   AxisStore[3].Axis[12].Pos24.Reached := FALSE;
   AxisStore[3].Axis[12].Pos25.Position := 0.0;
   AxisStore[3].Axis[12].Pos25.Speed := 0;
   AxisStore[3].Axis[12].Pos25.Reached := FALSE;
   AxisStore[3].Axis[12].Pos26.Position := 0.0;
   AxisStore[3].Axis[12].Pos26.Speed := 0;
   AxisStore[3].Axis[12].Pos26.Reached := FALSE;
   AxisStore[3].Axis[12].Pos27.Position := 0.0;
   AxisStore[3].Axis[12].Pos27.Speed := 0;
   AxisStore[3].Axis[12].Pos27.Reached := FALSE;
   AxisStore[3].Axis[12].Pos28.Position := 0.0;
   AxisStore[3].Axis[12].Pos28.Speed := 0;
   AxisStore[3].Axis[12].Pos28.Reached := FALSE;
   AxisStore[3].Axis[12].Pos29.Position := 0.0;
   AxisStore[3].Axis[12].Pos29.Speed := 0;
   AxisStore[3].Axis[12].Pos29.Reached := FALSE;
   AxisStore[3].Axis[12].Pos30.Position := 0.0;
   AxisStore[3].Axis[12].Pos30.Speed := 0;
   AxisStore[3].Axis[12].Pos30.Reached := FALSE;
   AxisStore[3].Axis[13].Pos1.Position := 0.0;
   AxisStore[3].Axis[13].Pos1.Speed := 0;
   AxisStore[3].Axis[13].Pos1.Reached := FALSE;
   AxisStore[3].Axis[13].Pos2.Position := 0.0;
   AxisStore[3].Axis[13].Pos2.Speed := 0;
   AxisStore[3].Axis[13].Pos2.Reached := FALSE;
   AxisStore[3].Axis[13].Pos3.Position := 0.0;
   AxisStore[3].Axis[13].Pos3.Speed := 0;
   AxisStore[3].Axis[13].Pos3.Reached := FALSE;
   AxisStore[3].Axis[13].Pos4.Position := 0.0;
   AxisStore[3].Axis[13].Pos4.Speed := 0;
   AxisStore[3].Axis[13].Pos4.Reached := FALSE;
   AxisStore[3].Axis[13].Pos5.Position := 0.0;
   AxisStore[3].Axis[13].Pos5.Speed := 0;
   AxisStore[3].Axis[13].Pos5.Reached := FALSE;
   AxisStore[3].Axis[13].Pos6.Position := 0.0;
   AxisStore[3].Axis[13].Pos6.Speed := 0;
   AxisStore[3].Axis[13].Pos6.Reached := FALSE;
   AxisStore[3].Axis[13].Pos7.Position := 0.0;
   AxisStore[3].Axis[13].Pos7.Speed := 0;
   AxisStore[3].Axis[13].Pos7.Reached := FALSE;
   AxisStore[3].Axis[13].Pos8.Position := 0.0;
   AxisStore[3].Axis[13].Pos8.Speed := 0;
   AxisStore[3].Axis[13].Pos8.Reached := FALSE;
   AxisStore[3].Axis[13].Pos9.Position := 0.0;
   AxisStore[3].Axis[13].Pos9.Speed := 0;
   AxisStore[3].Axis[13].Pos9.Reached := FALSE;
   AxisStore[3].Axis[13].Pos10.Position := 0.0;
   AxisStore[3].Axis[13].Pos10.Speed := 0;
   AxisStore[3].Axis[13].Pos10.Reached := FALSE;
   AxisStore[3].Axis[13].Pos11.Position := 0.0;
   AxisStore[3].Axis[13].Pos11.Speed := 0;
   AxisStore[3].Axis[13].Pos11.Reached := FALSE;
   AxisStore[3].Axis[13].Pos12.Position := 0.0;
   AxisStore[3].Axis[13].Pos12.Speed := 0;
   AxisStore[3].Axis[13].Pos12.Reached := FALSE;
   AxisStore[3].Axis[13].Pos13.Position := 0.0;
   AxisStore[3].Axis[13].Pos13.Speed := 0;
   AxisStore[3].Axis[13].Pos13.Reached := FALSE;
   AxisStore[3].Axis[13].Pos14.Position := 0.0;
   AxisStore[3].Axis[13].Pos14.Speed := 0;
   AxisStore[3].Axis[13].Pos14.Reached := FALSE;
   AxisStore[3].Axis[13].Pos15.Position := 0.0;
   AxisStore[3].Axis[13].Pos15.Speed := 0;
   AxisStore[3].Axis[13].Pos15.Reached := FALSE;
   AxisStore[3].Axis[13].Pos16.Position := 0.0;
   AxisStore[3].Axis[13].Pos16.Speed := 0;
   AxisStore[3].Axis[13].Pos16.Reached := FALSE;
   AxisStore[3].Axis[13].Pos17.Position := 0.0;
   AxisStore[3].Axis[13].Pos17.Speed := 0;
   AxisStore[3].Axis[13].Pos17.Reached := FALSE;
   AxisStore[3].Axis[13].Pos18.Position := 0.0;
   AxisStore[3].Axis[13].Pos18.Speed := 0;
   AxisStore[3].Axis[13].Pos18.Reached := FALSE;
   AxisStore[3].Axis[13].Pos19.Position := 0.0;
   AxisStore[3].Axis[13].Pos19.Speed := 0;
   AxisStore[3].Axis[13].Pos19.Reached := FALSE;
   AxisStore[3].Axis[13].Pos20.Position := 0.0;
   AxisStore[3].Axis[13].Pos20.Speed := 0;
   AxisStore[3].Axis[13].Pos20.Reached := FALSE;
   AxisStore[3].Axis[13].Pos21.Position := 0.0;
   AxisStore[3].Axis[13].Pos21.Speed := 0;
   AxisStore[3].Axis[13].Pos21.Reached := FALSE;
   AxisStore[3].Axis[13].Pos22.Position := 0.0;
   AxisStore[3].Axis[13].Pos22.Speed := 0;
   AxisStore[3].Axis[13].Pos22.Reached := FALSE;
   AxisStore[3].Axis[13].Pos23.Position := 0.0;
   AxisStore[3].Axis[13].Pos23.Speed := 0;
   AxisStore[3].Axis[13].Pos23.Reached := FALSE;
   AxisStore[3].Axis[13].Pos24.Position := 0.0;
   AxisStore[3].Axis[13].Pos24.Speed := 0;
   AxisStore[3].Axis[13].Pos24.Reached := FALSE;
   AxisStore[3].Axis[13].Pos25.Position := 0.0;
   AxisStore[3].Axis[13].Pos25.Speed := 0;
   AxisStore[3].Axis[13].Pos25.Reached := FALSE;
   AxisStore[3].Axis[13].Pos26.Position := 0.0;
   AxisStore[3].Axis[13].Pos26.Speed := 0;
   AxisStore[3].Axis[13].Pos26.Reached := FALSE;
   AxisStore[3].Axis[13].Pos27.Position := 0.0;
   AxisStore[3].Axis[13].Pos27.Speed := 0;
   AxisStore[3].Axis[13].Pos27.Reached := FALSE;
   AxisStore[3].Axis[13].Pos28.Position := 0.0;
   AxisStore[3].Axis[13].Pos28.Speed := 0;
   AxisStore[3].Axis[13].Pos28.Reached := FALSE;
   AxisStore[3].Axis[13].Pos29.Position := 0.0;
   AxisStore[3].Axis[13].Pos29.Speed := 0;
   AxisStore[3].Axis[13].Pos29.Reached := FALSE;
   AxisStore[3].Axis[13].Pos30.Position := 0.0;
   AxisStore[3].Axis[13].Pos30.Speed := 0;
   AxisStore[3].Axis[13].Pos30.Reached := FALSE;
   AxisStore[3].Axis[14].Pos1.Position := 0.0;
   AxisStore[3].Axis[14].Pos1.Speed := 0;
   AxisStore[3].Axis[14].Pos1.Reached := FALSE;
   AxisStore[3].Axis[14].Pos2.Position := 0.0;
   AxisStore[3].Axis[14].Pos2.Speed := 0;
   AxisStore[3].Axis[14].Pos2.Reached := FALSE;
   AxisStore[3].Axis[14].Pos3.Position := 0.0;
   AxisStore[3].Axis[14].Pos3.Speed := 0;
   AxisStore[3].Axis[14].Pos3.Reached := FALSE;
   AxisStore[3].Axis[14].Pos4.Position := 0.0;
   AxisStore[3].Axis[14].Pos4.Speed := 0;
   AxisStore[3].Axis[14].Pos4.Reached := FALSE;
   AxisStore[3].Axis[14].Pos5.Position := 0.0;
   AxisStore[3].Axis[14].Pos5.Speed := 0;
   AxisStore[3].Axis[14].Pos5.Reached := FALSE;
   AxisStore[3].Axis[14].Pos6.Position := 0.0;
   AxisStore[3].Axis[14].Pos6.Speed := 0;
   AxisStore[3].Axis[14].Pos6.Reached := FALSE;
   AxisStore[3].Axis[14].Pos7.Position := 0.0;
   AxisStore[3].Axis[14].Pos7.Speed := 0;
   AxisStore[3].Axis[14].Pos7.Reached := FALSE;
   AxisStore[3].Axis[14].Pos8.Position := 0.0;
   AxisStore[3].Axis[14].Pos8.Speed := 0;
   AxisStore[3].Axis[14].Pos8.Reached := FALSE;
   AxisStore[3].Axis[14].Pos9.Position := 0.0;
   AxisStore[3].Axis[14].Pos9.Speed := 0;
   AxisStore[3].Axis[14].Pos9.Reached := FALSE;
   AxisStore[3].Axis[14].Pos10.Position := 0.0;
   AxisStore[3].Axis[14].Pos10.Speed := 0;
   AxisStore[3].Axis[14].Pos10.Reached := FALSE;
   AxisStore[3].Axis[14].Pos11.Position := 0.0;
   AxisStore[3].Axis[14].Pos11.Speed := 0;
   AxisStore[3].Axis[14].Pos11.Reached := FALSE;
   AxisStore[3].Axis[14].Pos12.Position := 0.0;
   AxisStore[3].Axis[14].Pos12.Speed := 0;
   AxisStore[3].Axis[14].Pos12.Reached := FALSE;
   AxisStore[3].Axis[14].Pos13.Position := 0.0;
   AxisStore[3].Axis[14].Pos13.Speed := 0;
   AxisStore[3].Axis[14].Pos13.Reached := FALSE;
   AxisStore[3].Axis[14].Pos14.Position := 0.0;
   AxisStore[3].Axis[14].Pos14.Speed := 0;
   AxisStore[3].Axis[14].Pos14.Reached := FALSE;
   AxisStore[3].Axis[14].Pos15.Position := 0.0;
   AxisStore[3].Axis[14].Pos15.Speed := 0;
   AxisStore[3].Axis[14].Pos15.Reached := FALSE;
   AxisStore[3].Axis[14].Pos16.Position := 0.0;
   AxisStore[3].Axis[14].Pos16.Speed := 0;
   AxisStore[3].Axis[14].Pos16.Reached := FALSE;
   AxisStore[3].Axis[14].Pos17.Position := 0.0;
   AxisStore[3].Axis[14].Pos17.Speed := 0;
   AxisStore[3].Axis[14].Pos17.Reached := FALSE;
   AxisStore[3].Axis[14].Pos18.Position := 0.0;
   AxisStore[3].Axis[14].Pos18.Speed := 0;
   AxisStore[3].Axis[14].Pos18.Reached := FALSE;
   AxisStore[3].Axis[14].Pos19.Position := 0.0;
   AxisStore[3].Axis[14].Pos19.Speed := 0;
   AxisStore[3].Axis[14].Pos19.Reached := FALSE;
   AxisStore[3].Axis[14].Pos20.Position := 0.0;
   AxisStore[3].Axis[14].Pos20.Speed := 0;
   AxisStore[3].Axis[14].Pos20.Reached := FALSE;
   AxisStore[3].Axis[14].Pos21.Position := 0.0;
   AxisStore[3].Axis[14].Pos21.Speed := 0;
   AxisStore[3].Axis[14].Pos21.Reached := FALSE;
   AxisStore[3].Axis[14].Pos22.Position := 0.0;
   AxisStore[3].Axis[14].Pos22.Speed := 0;
   AxisStore[3].Axis[14].Pos22.Reached := FALSE;
   AxisStore[3].Axis[14].Pos23.Position := 0.0;
   AxisStore[3].Axis[14].Pos23.Speed := 0;
   AxisStore[3].Axis[14].Pos23.Reached := FALSE;
   AxisStore[3].Axis[14].Pos24.Position := 0.0;
   AxisStore[3].Axis[14].Pos24.Speed := 0;
   AxisStore[3].Axis[14].Pos24.Reached := FALSE;
   AxisStore[3].Axis[14].Pos25.Position := 0.0;
   AxisStore[3].Axis[14].Pos25.Speed := 0;
   AxisStore[3].Axis[14].Pos25.Reached := FALSE;
   AxisStore[3].Axis[14].Pos26.Position := 0.0;
   AxisStore[3].Axis[14].Pos26.Speed := 0;
   AxisStore[3].Axis[14].Pos26.Reached := FALSE;
   AxisStore[3].Axis[14].Pos27.Position := 0.0;
   AxisStore[3].Axis[14].Pos27.Speed := 0;
   AxisStore[3].Axis[14].Pos27.Reached := FALSE;
   AxisStore[3].Axis[14].Pos28.Position := 0.0;
   AxisStore[3].Axis[14].Pos28.Speed := 0;
   AxisStore[3].Axis[14].Pos28.Reached := FALSE;
   AxisStore[3].Axis[14].Pos29.Position := 0.0;
   AxisStore[3].Axis[14].Pos29.Speed := 0;
   AxisStore[3].Axis[14].Pos29.Reached := FALSE;
   AxisStore[3].Axis[14].Pos30.Position := 0.0;
   AxisStore[3].Axis[14].Pos30.Speed := 0;
   AxisStore[3].Axis[14].Pos30.Reached := FALSE;
   AxisStore[3].Axis[15].Pos1.Position := 0.0;
   AxisStore[3].Axis[15].Pos1.Speed := 0;
   AxisStore[3].Axis[15].Pos1.Reached := FALSE;
   AxisStore[3].Axis[15].Pos2.Position := 0.0;
   AxisStore[3].Axis[15].Pos2.Speed := 0;
   AxisStore[3].Axis[15].Pos2.Reached := FALSE;
   AxisStore[3].Axis[15].Pos3.Position := 0.0;
   AxisStore[3].Axis[15].Pos3.Speed := 0;
   AxisStore[3].Axis[15].Pos3.Reached := FALSE;
   AxisStore[3].Axis[15].Pos4.Position := 0.0;
   AxisStore[3].Axis[15].Pos4.Speed := 0;
   AxisStore[3].Axis[15].Pos4.Reached := FALSE;
   AxisStore[3].Axis[15].Pos5.Position := 0.0;
   AxisStore[3].Axis[15].Pos5.Speed := 0;
   AxisStore[3].Axis[15].Pos5.Reached := FALSE;
   AxisStore[3].Axis[15].Pos6.Position := 0.0;
   AxisStore[3].Axis[15].Pos6.Speed := 0;
   AxisStore[3].Axis[15].Pos6.Reached := FALSE;
   AxisStore[3].Axis[15].Pos7.Position := 0.0;
   AxisStore[3].Axis[15].Pos7.Speed := 0;
   AxisStore[3].Axis[15].Pos7.Reached := FALSE;
   AxisStore[3].Axis[15].Pos8.Position := 0.0;
   AxisStore[3].Axis[15].Pos8.Speed := 0;
   AxisStore[3].Axis[15].Pos8.Reached := FALSE;
   AxisStore[3].Axis[15].Pos9.Position := 0.0;
   AxisStore[3].Axis[15].Pos9.Speed := 0;
   AxisStore[3].Axis[15].Pos9.Reached := FALSE;
   AxisStore[3].Axis[15].Pos10.Position := 0.0;
   AxisStore[3].Axis[15].Pos10.Speed := 0;
   AxisStore[3].Axis[15].Pos10.Reached := FALSE;
   AxisStore[3].Axis[15].Pos11.Position := 0.0;
   AxisStore[3].Axis[15].Pos11.Speed := 0;
   AxisStore[3].Axis[15].Pos11.Reached := FALSE;
   AxisStore[3].Axis[15].Pos12.Position := 0.0;
   AxisStore[3].Axis[15].Pos12.Speed := 0;
   AxisStore[3].Axis[15].Pos12.Reached := FALSE;
   AxisStore[3].Axis[15].Pos13.Position := 0.0;
   AxisStore[3].Axis[15].Pos13.Speed := 0;
   AxisStore[3].Axis[15].Pos13.Reached := FALSE;
   AxisStore[3].Axis[15].Pos14.Position := 0.0;
   AxisStore[3].Axis[15].Pos14.Speed := 0;
   AxisStore[3].Axis[15].Pos14.Reached := FALSE;
   AxisStore[3].Axis[15].Pos15.Position := 0.0;
   AxisStore[3].Axis[15].Pos15.Speed := 0;
   AxisStore[3].Axis[15].Pos15.Reached := FALSE;
   AxisStore[3].Axis[15].Pos16.Position := 0.0;
   AxisStore[3].Axis[15].Pos16.Speed := 0;
   AxisStore[3].Axis[15].Pos16.Reached := FALSE;
   AxisStore[3].Axis[15].Pos17.Position := 0.0;
   AxisStore[3].Axis[15].Pos17.Speed := 0;
   AxisStore[3].Axis[15].Pos17.Reached := FALSE;
   AxisStore[3].Axis[15].Pos18.Position := 0.0;
   AxisStore[3].Axis[15].Pos18.Speed := 0;
   AxisStore[3].Axis[15].Pos18.Reached := FALSE;
   AxisStore[3].Axis[15].Pos19.Position := 0.0;
   AxisStore[3].Axis[15].Pos19.Speed := 0;
   AxisStore[3].Axis[15].Pos19.Reached := FALSE;
   AxisStore[3].Axis[15].Pos20.Position := 0.0;
   AxisStore[3].Axis[15].Pos20.Speed := 0;
   AxisStore[3].Axis[15].Pos20.Reached := FALSE;
   AxisStore[3].Axis[15].Pos21.Position := 0.0;
   AxisStore[3].Axis[15].Pos21.Speed := 0;
   AxisStore[3].Axis[15].Pos21.Reached := FALSE;
   AxisStore[3].Axis[15].Pos22.Position := 0.0;
   AxisStore[3].Axis[15].Pos22.Speed := 0;
   AxisStore[3].Axis[15].Pos22.Reached := FALSE;
   AxisStore[3].Axis[15].Pos23.Position := 0.0;
   AxisStore[3].Axis[15].Pos23.Speed := 0;
   AxisStore[3].Axis[15].Pos23.Reached := FALSE;
   AxisStore[3].Axis[15].Pos24.Position := 0.0;
   AxisStore[3].Axis[15].Pos24.Speed := 0;
   AxisStore[3].Axis[15].Pos24.Reached := FALSE;
   AxisStore[3].Axis[15].Pos25.Position := 0.0;
   AxisStore[3].Axis[15].Pos25.Speed := 0;
   AxisStore[3].Axis[15].Pos25.Reached := FALSE;
   AxisStore[3].Axis[15].Pos26.Position := 0.0;
   AxisStore[3].Axis[15].Pos26.Speed := 0;
   AxisStore[3].Axis[15].Pos26.Reached := FALSE;
   AxisStore[3].Axis[15].Pos27.Position := 0.0;
   AxisStore[3].Axis[15].Pos27.Speed := 0;
   AxisStore[3].Axis[15].Pos27.Reached := FALSE;
   AxisStore[3].Axis[15].Pos28.Position := 0.0;
   AxisStore[3].Axis[15].Pos28.Speed := 0;
   AxisStore[3].Axis[15].Pos28.Reached := FALSE;
   AxisStore[3].Axis[15].Pos29.Position := 0.0;
   AxisStore[3].Axis[15].Pos29.Speed := 0;
   AxisStore[3].Axis[15].Pos29.Reached := FALSE;
   AxisStore[3].Axis[15].Pos30.Position := 0.0;
   AxisStore[3].Axis[15].Pos30.Speed := 0;
   AxisStore[3].Axis[15].Pos30.Reached := FALSE;
   AxisStore[4].Axis[1].Pos1.Position := 0.0;
   AxisStore[4].Axis[1].Pos1.Speed := 0;
   AxisStore[4].Axis[1].Pos1.Reached := FALSE;
   AxisStore[4].Axis[1].Pos2.Position := 0.0;
   AxisStore[4].Axis[1].Pos2.Speed := 0;
   AxisStore[4].Axis[1].Pos2.Reached := FALSE;
   AxisStore[4].Axis[1].Pos3.Position := 0.0;
   AxisStore[4].Axis[1].Pos3.Speed := 0;
   AxisStore[4].Axis[1].Pos3.Reached := FALSE;
   AxisStore[4].Axis[1].Pos4.Position := 0.0;
   AxisStore[4].Axis[1].Pos4.Speed := 0;
   AxisStore[4].Axis[1].Pos4.Reached := FALSE;
   AxisStore[4].Axis[1].Pos5.Position := 0.0;
   AxisStore[4].Axis[1].Pos5.Speed := 0;
   AxisStore[4].Axis[1].Pos5.Reached := FALSE;
   AxisStore[4].Axis[1].Pos6.Position := 0.0;
   AxisStore[4].Axis[1].Pos6.Speed := 0;
   AxisStore[4].Axis[1].Pos6.Reached := FALSE;
   AxisStore[4].Axis[1].Pos7.Position := 0.0;
   AxisStore[4].Axis[1].Pos7.Speed := 0;
   AxisStore[4].Axis[1].Pos7.Reached := FALSE;
   AxisStore[4].Axis[1].Pos8.Position := 0.0;
   AxisStore[4].Axis[1].Pos8.Speed := 0;
   AxisStore[4].Axis[1].Pos8.Reached := FALSE;
   AxisStore[4].Axis[1].Pos9.Position := 0.0;
   AxisStore[4].Axis[1].Pos9.Speed := 0;
   AxisStore[4].Axis[1].Pos9.Reached := FALSE;
   AxisStore[4].Axis[1].Pos10.Position := 0.0;
   AxisStore[4].Axis[1].Pos10.Speed := 0;
   AxisStore[4].Axis[1].Pos10.Reached := FALSE;
   AxisStore[4].Axis[1].Pos11.Position := 0.0;
   AxisStore[4].Axis[1].Pos11.Speed := 0;
   AxisStore[4].Axis[1].Pos11.Reached := FALSE;
   AxisStore[4].Axis[1].Pos12.Position := 0.0;
   AxisStore[4].Axis[1].Pos12.Speed := 0;
   AxisStore[4].Axis[1].Pos12.Reached := FALSE;
   AxisStore[4].Axis[1].Pos13.Position := 0.0;
   AxisStore[4].Axis[1].Pos13.Speed := 0;
   AxisStore[4].Axis[1].Pos13.Reached := FALSE;
   AxisStore[4].Axis[1].Pos14.Position := 0.0;
   AxisStore[4].Axis[1].Pos14.Speed := 0;
   AxisStore[4].Axis[1].Pos14.Reached := FALSE;
   AxisStore[4].Axis[1].Pos15.Position := 0.0;
   AxisStore[4].Axis[1].Pos15.Speed := 0;
   AxisStore[4].Axis[1].Pos15.Reached := FALSE;
   AxisStore[4].Axis[1].Pos16.Position := 0.0;
   AxisStore[4].Axis[1].Pos16.Speed := 0;
   AxisStore[4].Axis[1].Pos16.Reached := FALSE;
   AxisStore[4].Axis[1].Pos17.Position := 0.0;
   AxisStore[4].Axis[1].Pos17.Speed := 0;
   AxisStore[4].Axis[1].Pos17.Reached := FALSE;
   AxisStore[4].Axis[1].Pos18.Position := 0.0;
   AxisStore[4].Axis[1].Pos18.Speed := 0;
   AxisStore[4].Axis[1].Pos18.Reached := FALSE;
   AxisStore[4].Axis[1].Pos19.Position := 0.0;
   AxisStore[4].Axis[1].Pos19.Speed := 0;
   AxisStore[4].Axis[1].Pos19.Reached := FALSE;
   AxisStore[4].Axis[1].Pos20.Position := 0.0;
   AxisStore[4].Axis[1].Pos20.Speed := 0;
   AxisStore[4].Axis[1].Pos20.Reached := FALSE;
   AxisStore[4].Axis[1].Pos21.Position := 0.0;
   AxisStore[4].Axis[1].Pos21.Speed := 0;
   AxisStore[4].Axis[1].Pos21.Reached := FALSE;
   AxisStore[4].Axis[1].Pos22.Position := 0.0;
   AxisStore[4].Axis[1].Pos22.Speed := 0;
   AxisStore[4].Axis[1].Pos22.Reached := FALSE;
   AxisStore[4].Axis[1].Pos23.Position := 0.0;
   AxisStore[4].Axis[1].Pos23.Speed := 0;
   AxisStore[4].Axis[1].Pos23.Reached := FALSE;
   AxisStore[4].Axis[1].Pos24.Position := 0.0;
   AxisStore[4].Axis[1].Pos24.Speed := 0;
   AxisStore[4].Axis[1].Pos24.Reached := FALSE;
   AxisStore[4].Axis[1].Pos25.Position := 0.0;
   AxisStore[4].Axis[1].Pos25.Speed := 0;
   AxisStore[4].Axis[1].Pos25.Reached := FALSE;
   AxisStore[4].Axis[1].Pos26.Position := 0.0;
   AxisStore[4].Axis[1].Pos26.Speed := 0;
   AxisStore[4].Axis[1].Pos26.Reached := FALSE;
   AxisStore[4].Axis[1].Pos27.Position := 0.0;
   AxisStore[4].Axis[1].Pos27.Speed := 0;
   AxisStore[4].Axis[1].Pos27.Reached := FALSE;
   AxisStore[4].Axis[1].Pos28.Position := 0.0;
   AxisStore[4].Axis[1].Pos28.Speed := 0;
   AxisStore[4].Axis[1].Pos28.Reached := FALSE;
   AxisStore[4].Axis[1].Pos29.Position := 0.0;
   AxisStore[4].Axis[1].Pos29.Speed := 0;
   AxisStore[4].Axis[1].Pos29.Reached := FALSE;
   AxisStore[4].Axis[1].Pos30.Position := 0.0;
   AxisStore[4].Axis[1].Pos30.Speed := 0;
   AxisStore[4].Axis[1].Pos30.Reached := FALSE;
   AxisStore[4].Axis[2].Pos1.Position := 0.0;
   AxisStore[4].Axis[2].Pos1.Speed := 0;
   AxisStore[4].Axis[2].Pos1.Reached := FALSE;
   AxisStore[4].Axis[2].Pos2.Position := 0.0;
   AxisStore[4].Axis[2].Pos2.Speed := 0;
   AxisStore[4].Axis[2].Pos2.Reached := FALSE;
   AxisStore[4].Axis[2].Pos3.Position := 0.0;
   AxisStore[4].Axis[2].Pos3.Speed := 0;
   AxisStore[4].Axis[2].Pos3.Reached := FALSE;
   AxisStore[4].Axis[2].Pos4.Position := 0.0;
   AxisStore[4].Axis[2].Pos4.Speed := 0;
   AxisStore[4].Axis[2].Pos4.Reached := FALSE;
   AxisStore[4].Axis[2].Pos5.Position := 0.0;
   AxisStore[4].Axis[2].Pos5.Speed := 0;
   AxisStore[4].Axis[2].Pos5.Reached := FALSE;
   AxisStore[4].Axis[2].Pos6.Position := 0.0;
   AxisStore[4].Axis[2].Pos6.Speed := 0;
   AxisStore[4].Axis[2].Pos6.Reached := FALSE;
   AxisStore[4].Axis[2].Pos7.Position := 0.0;
   AxisStore[4].Axis[2].Pos7.Speed := 0;
   AxisStore[4].Axis[2].Pos7.Reached := FALSE;
   AxisStore[4].Axis[2].Pos8.Position := 0.0;
   AxisStore[4].Axis[2].Pos8.Speed := 0;
   AxisStore[4].Axis[2].Pos8.Reached := FALSE;
   AxisStore[4].Axis[2].Pos9.Position := 0.0;
   AxisStore[4].Axis[2].Pos9.Speed := 0;
   AxisStore[4].Axis[2].Pos9.Reached := FALSE;
   AxisStore[4].Axis[2].Pos10.Position := 0.0;
   AxisStore[4].Axis[2].Pos10.Speed := 0;
   AxisStore[4].Axis[2].Pos10.Reached := FALSE;
   AxisStore[4].Axis[2].Pos11.Position := 0.0;
   AxisStore[4].Axis[2].Pos11.Speed := 0;
   AxisStore[4].Axis[2].Pos11.Reached := FALSE;
   AxisStore[4].Axis[2].Pos12.Position := 0.0;
   AxisStore[4].Axis[2].Pos12.Speed := 0;
   AxisStore[4].Axis[2].Pos12.Reached := FALSE;
   AxisStore[4].Axis[2].Pos13.Position := 0.0;
   AxisStore[4].Axis[2].Pos13.Speed := 0;
   AxisStore[4].Axis[2].Pos13.Reached := FALSE;
   AxisStore[4].Axis[2].Pos14.Position := 0.0;
   AxisStore[4].Axis[2].Pos14.Speed := 0;
   AxisStore[4].Axis[2].Pos14.Reached := FALSE;
   AxisStore[4].Axis[2].Pos15.Position := 0.0;
   AxisStore[4].Axis[2].Pos15.Speed := 0;
   AxisStore[4].Axis[2].Pos15.Reached := FALSE;
   AxisStore[4].Axis[2].Pos16.Position := 0.0;
   AxisStore[4].Axis[2].Pos16.Speed := 0;
   AxisStore[4].Axis[2].Pos16.Reached := FALSE;
   AxisStore[4].Axis[2].Pos17.Position := 0.0;
   AxisStore[4].Axis[2].Pos17.Speed := 0;
   AxisStore[4].Axis[2].Pos17.Reached := FALSE;
   AxisStore[4].Axis[2].Pos18.Position := 0.0;
   AxisStore[4].Axis[2].Pos18.Speed := 0;
   AxisStore[4].Axis[2].Pos18.Reached := FALSE;
   AxisStore[4].Axis[2].Pos19.Position := 0.0;
   AxisStore[4].Axis[2].Pos19.Speed := 0;
   AxisStore[4].Axis[2].Pos19.Reached := FALSE;
   AxisStore[4].Axis[2].Pos20.Position := 0.0;
   AxisStore[4].Axis[2].Pos20.Speed := 0;
   AxisStore[4].Axis[2].Pos20.Reached := FALSE;
   AxisStore[4].Axis[2].Pos21.Position := 0.0;
   AxisStore[4].Axis[2].Pos21.Speed := 0;
   AxisStore[4].Axis[2].Pos21.Reached := FALSE;
   AxisStore[4].Axis[2].Pos22.Position := 0.0;
   AxisStore[4].Axis[2].Pos22.Speed := 0;
   AxisStore[4].Axis[2].Pos22.Reached := FALSE;
   AxisStore[4].Axis[2].Pos23.Position := 0.0;
   AxisStore[4].Axis[2].Pos23.Speed := 0;
   AxisStore[4].Axis[2].Pos23.Reached := FALSE;
   AxisStore[4].Axis[2].Pos24.Position := 0.0;
   AxisStore[4].Axis[2].Pos24.Speed := 0;
   AxisStore[4].Axis[2].Pos24.Reached := FALSE;
   AxisStore[4].Axis[2].Pos25.Position := 0.0;
   AxisStore[4].Axis[2].Pos25.Speed := 0;
   AxisStore[4].Axis[2].Pos25.Reached := FALSE;
   AxisStore[4].Axis[2].Pos26.Position := 0.0;
   AxisStore[4].Axis[2].Pos26.Speed := 0;
   AxisStore[4].Axis[2].Pos26.Reached := FALSE;
   AxisStore[4].Axis[2].Pos27.Position := 0.0;
   AxisStore[4].Axis[2].Pos27.Speed := 0;
   AxisStore[4].Axis[2].Pos27.Reached := FALSE;
   AxisStore[4].Axis[2].Pos28.Position := 0.0;
   AxisStore[4].Axis[2].Pos28.Speed := 0;
   AxisStore[4].Axis[2].Pos28.Reached := FALSE;
   AxisStore[4].Axis[2].Pos29.Position := 0.0;
   AxisStore[4].Axis[2].Pos29.Speed := 0;
   AxisStore[4].Axis[2].Pos29.Reached := FALSE;
   AxisStore[4].Axis[2].Pos30.Position := 0.0;
   AxisStore[4].Axis[2].Pos30.Speed := 0;
   AxisStore[4].Axis[2].Pos30.Reached := FALSE;
   AxisStore[4].Axis[3].Pos1.Position := 0.0;
   AxisStore[4].Axis[3].Pos1.Speed := 0;
   AxisStore[4].Axis[3].Pos1.Reached := FALSE;
   AxisStore[4].Axis[3].Pos2.Position := 0.0;
   AxisStore[4].Axis[3].Pos2.Speed := 0;
   AxisStore[4].Axis[3].Pos2.Reached := FALSE;
   AxisStore[4].Axis[3].Pos3.Position := 0.0;
   AxisStore[4].Axis[3].Pos3.Speed := 0;
   AxisStore[4].Axis[3].Pos3.Reached := FALSE;
   AxisStore[4].Axis[3].Pos4.Position := 0.0;
   AxisStore[4].Axis[3].Pos4.Speed := 0;
   AxisStore[4].Axis[3].Pos4.Reached := FALSE;
   AxisStore[4].Axis[3].Pos5.Position := 0.0;
   AxisStore[4].Axis[3].Pos5.Speed := 0;
   AxisStore[4].Axis[3].Pos5.Reached := FALSE;
   AxisStore[4].Axis[3].Pos6.Position := 0.0;
   AxisStore[4].Axis[3].Pos6.Speed := 0;
   AxisStore[4].Axis[3].Pos6.Reached := FALSE;
   AxisStore[4].Axis[3].Pos7.Position := 0.0;
   AxisStore[4].Axis[3].Pos7.Speed := 0;
   AxisStore[4].Axis[3].Pos7.Reached := FALSE;
   AxisStore[4].Axis[3].Pos8.Position := 0.0;
   AxisStore[4].Axis[3].Pos8.Speed := 0;
   AxisStore[4].Axis[3].Pos8.Reached := FALSE;
   AxisStore[4].Axis[3].Pos9.Position := 0.0;
   AxisStore[4].Axis[3].Pos9.Speed := 0;
   AxisStore[4].Axis[3].Pos9.Reached := FALSE;
   AxisStore[4].Axis[3].Pos10.Position := 0.0;
   AxisStore[4].Axis[3].Pos10.Speed := 0;
   AxisStore[4].Axis[3].Pos10.Reached := FALSE;
   AxisStore[4].Axis[3].Pos11.Position := 0.0;
   AxisStore[4].Axis[3].Pos11.Speed := 0;
   AxisStore[4].Axis[3].Pos11.Reached := FALSE;
   AxisStore[4].Axis[3].Pos12.Position := 0.0;
   AxisStore[4].Axis[3].Pos12.Speed := 0;
   AxisStore[4].Axis[3].Pos12.Reached := FALSE;
   AxisStore[4].Axis[3].Pos13.Position := 0.0;
   AxisStore[4].Axis[3].Pos13.Speed := 0;
   AxisStore[4].Axis[3].Pos13.Reached := FALSE;
   AxisStore[4].Axis[3].Pos14.Position := 0.0;
   AxisStore[4].Axis[3].Pos14.Speed := 0;
   AxisStore[4].Axis[3].Pos14.Reached := FALSE;
   AxisStore[4].Axis[3].Pos15.Position := 0.0;
   AxisStore[4].Axis[3].Pos15.Speed := 0;
   AxisStore[4].Axis[3].Pos15.Reached := FALSE;
   AxisStore[4].Axis[3].Pos16.Position := 0.0;
   AxisStore[4].Axis[3].Pos16.Speed := 0;
   AxisStore[4].Axis[3].Pos16.Reached := FALSE;
   AxisStore[4].Axis[3].Pos17.Position := 0.0;
   AxisStore[4].Axis[3].Pos17.Speed := 0;
   AxisStore[4].Axis[3].Pos17.Reached := FALSE;
   AxisStore[4].Axis[3].Pos18.Position := 0.0;
   AxisStore[4].Axis[3].Pos18.Speed := 0;
   AxisStore[4].Axis[3].Pos18.Reached := FALSE;
   AxisStore[4].Axis[3].Pos19.Position := 0.0;
   AxisStore[4].Axis[3].Pos19.Speed := 0;
   AxisStore[4].Axis[3].Pos19.Reached := FALSE;
   AxisStore[4].Axis[3].Pos20.Position := 0.0;
   AxisStore[4].Axis[3].Pos20.Speed := 0;
   AxisStore[4].Axis[3].Pos20.Reached := FALSE;
   AxisStore[4].Axis[3].Pos21.Position := 0.0;
   AxisStore[4].Axis[3].Pos21.Speed := 0;
   AxisStore[4].Axis[3].Pos21.Reached := FALSE;
   AxisStore[4].Axis[3].Pos22.Position := 0.0;
   AxisStore[4].Axis[3].Pos22.Speed := 0;
   AxisStore[4].Axis[3].Pos22.Reached := FALSE;
   AxisStore[4].Axis[3].Pos23.Position := 0.0;
   AxisStore[4].Axis[3].Pos23.Speed := 0;
   AxisStore[4].Axis[3].Pos23.Reached := FALSE;
   AxisStore[4].Axis[3].Pos24.Position := 0.0;
   AxisStore[4].Axis[3].Pos24.Speed := 0;
   AxisStore[4].Axis[3].Pos24.Reached := FALSE;
   AxisStore[4].Axis[3].Pos25.Position := 0.0;
   AxisStore[4].Axis[3].Pos25.Speed := 0;
   AxisStore[4].Axis[3].Pos25.Reached := FALSE;
   AxisStore[4].Axis[3].Pos26.Position := 0.0;
   AxisStore[4].Axis[3].Pos26.Speed := 0;
   AxisStore[4].Axis[3].Pos26.Reached := FALSE;
   AxisStore[4].Axis[3].Pos27.Position := 0.0;
   AxisStore[4].Axis[3].Pos27.Speed := 0;
   AxisStore[4].Axis[3].Pos27.Reached := FALSE;
   AxisStore[4].Axis[3].Pos28.Position := 0.0;
   AxisStore[4].Axis[3].Pos28.Speed := 0;
   AxisStore[4].Axis[3].Pos28.Reached := FALSE;
   AxisStore[4].Axis[3].Pos29.Position := 0.0;
   AxisStore[4].Axis[3].Pos29.Speed := 0;
   AxisStore[4].Axis[3].Pos29.Reached := FALSE;
   AxisStore[4].Axis[3].Pos30.Position := 0.0;
   AxisStore[4].Axis[3].Pos30.Speed := 0;
   AxisStore[4].Axis[3].Pos30.Reached := FALSE;
   AxisStore[4].Axis[4].Pos1.Position := 0.0;
   AxisStore[4].Axis[4].Pos1.Speed := 0;
   AxisStore[4].Axis[4].Pos1.Reached := FALSE;
   AxisStore[4].Axis[4].Pos2.Position := 0.0;
   AxisStore[4].Axis[4].Pos2.Speed := 0;
   AxisStore[4].Axis[4].Pos2.Reached := FALSE;
   AxisStore[4].Axis[4].Pos3.Position := 0.0;
   AxisStore[4].Axis[4].Pos3.Speed := 0;
   AxisStore[4].Axis[4].Pos3.Reached := FALSE;
   AxisStore[4].Axis[4].Pos4.Position := 0.0;
   AxisStore[4].Axis[4].Pos4.Speed := 0;
   AxisStore[4].Axis[4].Pos4.Reached := FALSE;
   AxisStore[4].Axis[4].Pos5.Position := 0.0;
   AxisStore[4].Axis[4].Pos5.Speed := 0;
   AxisStore[4].Axis[4].Pos5.Reached := FALSE;
   AxisStore[4].Axis[4].Pos6.Position := 0.0;
   AxisStore[4].Axis[4].Pos6.Speed := 0;
   AxisStore[4].Axis[4].Pos6.Reached := FALSE;
   AxisStore[4].Axis[4].Pos7.Position := 0.0;
   AxisStore[4].Axis[4].Pos7.Speed := 0;
   AxisStore[4].Axis[4].Pos7.Reached := FALSE;
   AxisStore[4].Axis[4].Pos8.Position := 0.0;
   AxisStore[4].Axis[4].Pos8.Speed := 0;
   AxisStore[4].Axis[4].Pos8.Reached := FALSE;
   AxisStore[4].Axis[4].Pos9.Position := 0.0;
   AxisStore[4].Axis[4].Pos9.Speed := 0;
   AxisStore[4].Axis[4].Pos9.Reached := FALSE;
   AxisStore[4].Axis[4].Pos10.Position := 0.0;
   AxisStore[4].Axis[4].Pos10.Speed := 0;
   AxisStore[4].Axis[4].Pos10.Reached := FALSE;
   AxisStore[4].Axis[4].Pos11.Position := 0.0;
   AxisStore[4].Axis[4].Pos11.Speed := 0;
   AxisStore[4].Axis[4].Pos11.Reached := FALSE;
   AxisStore[4].Axis[4].Pos12.Position := 0.0;
   AxisStore[4].Axis[4].Pos12.Speed := 0;
   AxisStore[4].Axis[4].Pos12.Reached := FALSE;
   AxisStore[4].Axis[4].Pos13.Position := 0.0;
   AxisStore[4].Axis[4].Pos13.Speed := 0;
   AxisStore[4].Axis[4].Pos13.Reached := FALSE;
   AxisStore[4].Axis[4].Pos14.Position := 0.0;
   AxisStore[4].Axis[4].Pos14.Speed := 0;
   AxisStore[4].Axis[4].Pos14.Reached := FALSE;
   AxisStore[4].Axis[4].Pos15.Position := 0.0;
   AxisStore[4].Axis[4].Pos15.Speed := 0;
   AxisStore[4].Axis[4].Pos15.Reached := FALSE;
   AxisStore[4].Axis[4].Pos16.Position := 0.0;
   AxisStore[4].Axis[4].Pos16.Speed := 0;
   AxisStore[4].Axis[4].Pos16.Reached := FALSE;
   AxisStore[4].Axis[4].Pos17.Position := 0.0;
   AxisStore[4].Axis[4].Pos17.Speed := 0;
   AxisStore[4].Axis[4].Pos17.Reached := FALSE;
   AxisStore[4].Axis[4].Pos18.Position := 0.0;
   AxisStore[4].Axis[4].Pos18.Speed := 0;
   AxisStore[4].Axis[4].Pos18.Reached := FALSE;
   AxisStore[4].Axis[4].Pos19.Position := 0.0;
   AxisStore[4].Axis[4].Pos19.Speed := 0;
   AxisStore[4].Axis[4].Pos19.Reached := FALSE;
   AxisStore[4].Axis[4].Pos20.Position := 0.0;
   AxisStore[4].Axis[4].Pos20.Speed := 0;
   AxisStore[4].Axis[4].Pos20.Reached := FALSE;
   AxisStore[4].Axis[4].Pos21.Position := 0.0;
   AxisStore[4].Axis[4].Pos21.Speed := 0;
   AxisStore[4].Axis[4].Pos21.Reached := FALSE;
   AxisStore[4].Axis[4].Pos22.Position := 0.0;
   AxisStore[4].Axis[4].Pos22.Speed := 0;
   AxisStore[4].Axis[4].Pos22.Reached := FALSE;
   AxisStore[4].Axis[4].Pos23.Position := 0.0;
   AxisStore[4].Axis[4].Pos23.Speed := 0;
   AxisStore[4].Axis[4].Pos23.Reached := FALSE;
   AxisStore[4].Axis[4].Pos24.Position := 0.0;
   AxisStore[4].Axis[4].Pos24.Speed := 0;
   AxisStore[4].Axis[4].Pos24.Reached := FALSE;
   AxisStore[4].Axis[4].Pos25.Position := 0.0;
   AxisStore[4].Axis[4].Pos25.Speed := 0;
   AxisStore[4].Axis[4].Pos25.Reached := FALSE;
   AxisStore[4].Axis[4].Pos26.Position := 0.0;
   AxisStore[4].Axis[4].Pos26.Speed := 0;
   AxisStore[4].Axis[4].Pos26.Reached := FALSE;
   AxisStore[4].Axis[4].Pos27.Position := 0.0;
   AxisStore[4].Axis[4].Pos27.Speed := 0;
   AxisStore[4].Axis[4].Pos27.Reached := FALSE;
   AxisStore[4].Axis[4].Pos28.Position := 0.0;
   AxisStore[4].Axis[4].Pos28.Speed := 0;
   AxisStore[4].Axis[4].Pos28.Reached := FALSE;
   AxisStore[4].Axis[4].Pos29.Position := 0.0;
   AxisStore[4].Axis[4].Pos29.Speed := 0;
   AxisStore[4].Axis[4].Pos29.Reached := FALSE;
   AxisStore[4].Axis[4].Pos30.Position := 0.0;
   AxisStore[4].Axis[4].Pos30.Speed := 0;
   AxisStore[4].Axis[4].Pos30.Reached := FALSE;
   AxisStore[4].Axis[5].Pos1.Position := 0.0;
   AxisStore[4].Axis[5].Pos1.Speed := 0;
   AxisStore[4].Axis[5].Pos1.Reached := FALSE;
   AxisStore[4].Axis[5].Pos2.Position := 0.0;
   AxisStore[4].Axis[5].Pos2.Speed := 0;
   AxisStore[4].Axis[5].Pos2.Reached := FALSE;
   AxisStore[4].Axis[5].Pos3.Position := 0.0;
   AxisStore[4].Axis[5].Pos3.Speed := 0;
   AxisStore[4].Axis[5].Pos3.Reached := FALSE;
   AxisStore[4].Axis[5].Pos4.Position := 0.0;
   AxisStore[4].Axis[5].Pos4.Speed := 0;
   AxisStore[4].Axis[5].Pos4.Reached := FALSE;
   AxisStore[4].Axis[5].Pos5.Position := 0.0;
   AxisStore[4].Axis[5].Pos5.Speed := 0;
   AxisStore[4].Axis[5].Pos5.Reached := FALSE;
   AxisStore[4].Axis[5].Pos6.Position := 0.0;
   AxisStore[4].Axis[5].Pos6.Speed := 0;
   AxisStore[4].Axis[5].Pos6.Reached := FALSE;
   AxisStore[4].Axis[5].Pos7.Position := 0.0;
   AxisStore[4].Axis[5].Pos7.Speed := 0;
   AxisStore[4].Axis[5].Pos7.Reached := FALSE;
   AxisStore[4].Axis[5].Pos8.Position := 0.0;
   AxisStore[4].Axis[5].Pos8.Speed := 0;
   AxisStore[4].Axis[5].Pos8.Reached := FALSE;
   AxisStore[4].Axis[5].Pos9.Position := 0.0;
   AxisStore[4].Axis[5].Pos9.Speed := 0;
   AxisStore[4].Axis[5].Pos9.Reached := FALSE;
   AxisStore[4].Axis[5].Pos10.Position := 0.0;
   AxisStore[4].Axis[5].Pos10.Speed := 0;
   AxisStore[4].Axis[5].Pos10.Reached := FALSE;
   AxisStore[4].Axis[5].Pos11.Position := 0.0;
   AxisStore[4].Axis[5].Pos11.Speed := 0;
   AxisStore[4].Axis[5].Pos11.Reached := FALSE;
   AxisStore[4].Axis[5].Pos12.Position := 0.0;
   AxisStore[4].Axis[5].Pos12.Speed := 0;
   AxisStore[4].Axis[5].Pos12.Reached := FALSE;
   AxisStore[4].Axis[5].Pos13.Position := 0.0;
   AxisStore[4].Axis[5].Pos13.Speed := 0;
   AxisStore[4].Axis[5].Pos13.Reached := FALSE;
   AxisStore[4].Axis[5].Pos14.Position := 0.0;
   AxisStore[4].Axis[5].Pos14.Speed := 0;
   AxisStore[4].Axis[5].Pos14.Reached := FALSE;
   AxisStore[4].Axis[5].Pos15.Position := 0.0;
   AxisStore[4].Axis[5].Pos15.Speed := 0;
   AxisStore[4].Axis[5].Pos15.Reached := FALSE;
   AxisStore[4].Axis[5].Pos16.Position := 0.0;
   AxisStore[4].Axis[5].Pos16.Speed := 0;
   AxisStore[4].Axis[5].Pos16.Reached := FALSE;
   AxisStore[4].Axis[5].Pos17.Position := 0.0;
   AxisStore[4].Axis[5].Pos17.Speed := 0;
   AxisStore[4].Axis[5].Pos17.Reached := FALSE;
   AxisStore[4].Axis[5].Pos18.Position := 0.0;
   AxisStore[4].Axis[5].Pos18.Speed := 0;
   AxisStore[4].Axis[5].Pos18.Reached := FALSE;
   AxisStore[4].Axis[5].Pos19.Position := 0.0;
   AxisStore[4].Axis[5].Pos19.Speed := 0;
   AxisStore[4].Axis[5].Pos19.Reached := FALSE;
   AxisStore[4].Axis[5].Pos20.Position := 0.0;
   AxisStore[4].Axis[5].Pos20.Speed := 0;
   AxisStore[4].Axis[5].Pos20.Reached := FALSE;
   AxisStore[4].Axis[5].Pos21.Position := 0.0;
   AxisStore[4].Axis[5].Pos21.Speed := 0;
   AxisStore[4].Axis[5].Pos21.Reached := FALSE;
   AxisStore[4].Axis[5].Pos22.Position := 0.0;
   AxisStore[4].Axis[5].Pos22.Speed := 0;
   AxisStore[4].Axis[5].Pos22.Reached := FALSE;
   AxisStore[4].Axis[5].Pos23.Position := 0.0;
   AxisStore[4].Axis[5].Pos23.Speed := 0;
   AxisStore[4].Axis[5].Pos23.Reached := FALSE;
   AxisStore[4].Axis[5].Pos24.Position := 0.0;
   AxisStore[4].Axis[5].Pos24.Speed := 0;
   AxisStore[4].Axis[5].Pos24.Reached := FALSE;
   AxisStore[4].Axis[5].Pos25.Position := 0.0;
   AxisStore[4].Axis[5].Pos25.Speed := 0;
   AxisStore[4].Axis[5].Pos25.Reached := FALSE;
   AxisStore[4].Axis[5].Pos26.Position := 0.0;
   AxisStore[4].Axis[5].Pos26.Speed := 0;
   AxisStore[4].Axis[5].Pos26.Reached := FALSE;
   AxisStore[4].Axis[5].Pos27.Position := 0.0;
   AxisStore[4].Axis[5].Pos27.Speed := 0;
   AxisStore[4].Axis[5].Pos27.Reached := FALSE;
   AxisStore[4].Axis[5].Pos28.Position := 0.0;
   AxisStore[4].Axis[5].Pos28.Speed := 0;
   AxisStore[4].Axis[5].Pos28.Reached := FALSE;
   AxisStore[4].Axis[5].Pos29.Position := 0.0;
   AxisStore[4].Axis[5].Pos29.Speed := 0;
   AxisStore[4].Axis[5].Pos29.Reached := FALSE;
   AxisStore[4].Axis[5].Pos30.Position := 0.0;
   AxisStore[4].Axis[5].Pos30.Speed := 0;
   AxisStore[4].Axis[5].Pos30.Reached := FALSE;
   AxisStore[4].Axis[6].Pos1.Position := 0.0;
   AxisStore[4].Axis[6].Pos1.Speed := 0;
   AxisStore[4].Axis[6].Pos1.Reached := FALSE;
   AxisStore[4].Axis[6].Pos2.Position := 0.0;
   AxisStore[4].Axis[6].Pos2.Speed := 0;
   AxisStore[4].Axis[6].Pos2.Reached := FALSE;
   AxisStore[4].Axis[6].Pos3.Position := 0.0;
   AxisStore[4].Axis[6].Pos3.Speed := 0;
   AxisStore[4].Axis[6].Pos3.Reached := FALSE;
   AxisStore[4].Axis[6].Pos4.Position := 0.0;
   AxisStore[4].Axis[6].Pos4.Speed := 0;
   AxisStore[4].Axis[6].Pos4.Reached := FALSE;
   AxisStore[4].Axis[6].Pos5.Position := 0.0;
   AxisStore[4].Axis[6].Pos5.Speed := 0;
   AxisStore[4].Axis[6].Pos5.Reached := FALSE;
   AxisStore[4].Axis[6].Pos6.Position := 0.0;
   AxisStore[4].Axis[6].Pos6.Speed := 0;
   AxisStore[4].Axis[6].Pos6.Reached := FALSE;
   AxisStore[4].Axis[6].Pos7.Position := 0.0;
   AxisStore[4].Axis[6].Pos7.Speed := 0;
   AxisStore[4].Axis[6].Pos7.Reached := FALSE;
   AxisStore[4].Axis[6].Pos8.Position := 0.0;
   AxisStore[4].Axis[6].Pos8.Speed := 0;
   AxisStore[4].Axis[6].Pos8.Reached := FALSE;
   AxisStore[4].Axis[6].Pos9.Position := 0.0;
   AxisStore[4].Axis[6].Pos9.Speed := 0;
   AxisStore[4].Axis[6].Pos9.Reached := FALSE;
   AxisStore[4].Axis[6].Pos10.Position := 0.0;
   AxisStore[4].Axis[6].Pos10.Speed := 0;
   AxisStore[4].Axis[6].Pos10.Reached := FALSE;
   AxisStore[4].Axis[6].Pos11.Position := 0.0;
   AxisStore[4].Axis[6].Pos11.Speed := 0;
   AxisStore[4].Axis[6].Pos11.Reached := FALSE;
   AxisStore[4].Axis[6].Pos12.Position := 0.0;
   AxisStore[4].Axis[6].Pos12.Speed := 0;
   AxisStore[4].Axis[6].Pos12.Reached := FALSE;
   AxisStore[4].Axis[6].Pos13.Position := 0.0;
   AxisStore[4].Axis[6].Pos13.Speed := 0;
   AxisStore[4].Axis[6].Pos13.Reached := FALSE;
   AxisStore[4].Axis[6].Pos14.Position := 0.0;
   AxisStore[4].Axis[6].Pos14.Speed := 0;
   AxisStore[4].Axis[6].Pos14.Reached := FALSE;
   AxisStore[4].Axis[6].Pos15.Position := 0.0;
   AxisStore[4].Axis[6].Pos15.Speed := 0;
   AxisStore[4].Axis[6].Pos15.Reached := FALSE;
   AxisStore[4].Axis[6].Pos16.Position := 0.0;
   AxisStore[4].Axis[6].Pos16.Speed := 0;
   AxisStore[4].Axis[6].Pos16.Reached := FALSE;
   AxisStore[4].Axis[6].Pos17.Position := 0.0;
   AxisStore[4].Axis[6].Pos17.Speed := 0;
   AxisStore[4].Axis[6].Pos17.Reached := FALSE;
   AxisStore[4].Axis[6].Pos18.Position := 0.0;
   AxisStore[4].Axis[6].Pos18.Speed := 0;
   AxisStore[4].Axis[6].Pos18.Reached := FALSE;
   AxisStore[4].Axis[6].Pos19.Position := 0.0;
   AxisStore[4].Axis[6].Pos19.Speed := 0;
   AxisStore[4].Axis[6].Pos19.Reached := FALSE;
   AxisStore[4].Axis[6].Pos20.Position := 0.0;
   AxisStore[4].Axis[6].Pos20.Speed := 0;
   AxisStore[4].Axis[6].Pos20.Reached := FALSE;
   AxisStore[4].Axis[6].Pos21.Position := 0.0;
   AxisStore[4].Axis[6].Pos21.Speed := 0;
   AxisStore[4].Axis[6].Pos21.Reached := FALSE;
   AxisStore[4].Axis[6].Pos22.Position := 0.0;
   AxisStore[4].Axis[6].Pos22.Speed := 0;
   AxisStore[4].Axis[6].Pos22.Reached := FALSE;
   AxisStore[4].Axis[6].Pos23.Position := 0.0;
   AxisStore[4].Axis[6].Pos23.Speed := 0;
   AxisStore[4].Axis[6].Pos23.Reached := FALSE;
   AxisStore[4].Axis[6].Pos24.Position := 0.0;
   AxisStore[4].Axis[6].Pos24.Speed := 0;
   AxisStore[4].Axis[6].Pos24.Reached := FALSE;
   AxisStore[4].Axis[6].Pos25.Position := 0.0;
   AxisStore[4].Axis[6].Pos25.Speed := 0;
   AxisStore[4].Axis[6].Pos25.Reached := FALSE;
   AxisStore[4].Axis[6].Pos26.Position := 0.0;
   AxisStore[4].Axis[6].Pos26.Speed := 0;
   AxisStore[4].Axis[6].Pos26.Reached := FALSE;
   AxisStore[4].Axis[6].Pos27.Position := 0.0;
   AxisStore[4].Axis[6].Pos27.Speed := 0;
   AxisStore[4].Axis[6].Pos27.Reached := FALSE;
   AxisStore[4].Axis[6].Pos28.Position := 0.0;
   AxisStore[4].Axis[6].Pos28.Speed := 0;
   AxisStore[4].Axis[6].Pos28.Reached := FALSE;
   AxisStore[4].Axis[6].Pos29.Position := 0.0;
   AxisStore[4].Axis[6].Pos29.Speed := 0;
   AxisStore[4].Axis[6].Pos29.Reached := FALSE;
   AxisStore[4].Axis[6].Pos30.Position := 0.0;
   AxisStore[4].Axis[6].Pos30.Speed := 0;
   AxisStore[4].Axis[6].Pos30.Reached := FALSE;
   AxisStore[4].Axis[7].Pos1.Position := 0.0;
   AxisStore[4].Axis[7].Pos1.Speed := 0;
   AxisStore[4].Axis[7].Pos1.Reached := FALSE;
   AxisStore[4].Axis[7].Pos2.Position := 0.0;
   AxisStore[4].Axis[7].Pos2.Speed := 0;
   AxisStore[4].Axis[7].Pos2.Reached := FALSE;
   AxisStore[4].Axis[7].Pos3.Position := 0.0;
   AxisStore[4].Axis[7].Pos3.Speed := 0;
   AxisStore[4].Axis[7].Pos3.Reached := FALSE;
   AxisStore[4].Axis[7].Pos4.Position := 0.0;
   AxisStore[4].Axis[7].Pos4.Speed := 0;
   AxisStore[4].Axis[7].Pos4.Reached := FALSE;
   AxisStore[4].Axis[7].Pos5.Position := 0.0;
   AxisStore[4].Axis[7].Pos5.Speed := 0;
   AxisStore[4].Axis[7].Pos5.Reached := FALSE;
   AxisStore[4].Axis[7].Pos6.Position := 0.0;
   AxisStore[4].Axis[7].Pos6.Speed := 0;
   AxisStore[4].Axis[7].Pos6.Reached := FALSE;
   AxisStore[4].Axis[7].Pos7.Position := 0.0;
   AxisStore[4].Axis[7].Pos7.Speed := 0;
   AxisStore[4].Axis[7].Pos7.Reached := FALSE;
   AxisStore[4].Axis[7].Pos8.Position := 0.0;
   AxisStore[4].Axis[7].Pos8.Speed := 0;
   AxisStore[4].Axis[7].Pos8.Reached := FALSE;
   AxisStore[4].Axis[7].Pos9.Position := 0.0;
   AxisStore[4].Axis[7].Pos9.Speed := 0;
   AxisStore[4].Axis[7].Pos9.Reached := FALSE;
   AxisStore[4].Axis[7].Pos10.Position := 0.0;
   AxisStore[4].Axis[7].Pos10.Speed := 0;
   AxisStore[4].Axis[7].Pos10.Reached := FALSE;
   AxisStore[4].Axis[7].Pos11.Position := 0.0;
   AxisStore[4].Axis[7].Pos11.Speed := 0;
   AxisStore[4].Axis[7].Pos11.Reached := FALSE;
   AxisStore[4].Axis[7].Pos12.Position := 0.0;
   AxisStore[4].Axis[7].Pos12.Speed := 0;
   AxisStore[4].Axis[7].Pos12.Reached := FALSE;
   AxisStore[4].Axis[7].Pos13.Position := 0.0;
   AxisStore[4].Axis[7].Pos13.Speed := 0;
   AxisStore[4].Axis[7].Pos13.Reached := FALSE;
   AxisStore[4].Axis[7].Pos14.Position := 0.0;
   AxisStore[4].Axis[7].Pos14.Speed := 0;
   AxisStore[4].Axis[7].Pos14.Reached := FALSE;
   AxisStore[4].Axis[7].Pos15.Position := 0.0;
   AxisStore[4].Axis[7].Pos15.Speed := 0;
   AxisStore[4].Axis[7].Pos15.Reached := FALSE;
   AxisStore[4].Axis[7].Pos16.Position := 0.0;
   AxisStore[4].Axis[7].Pos16.Speed := 0;
   AxisStore[4].Axis[7].Pos16.Reached := FALSE;
   AxisStore[4].Axis[7].Pos17.Position := 0.0;
   AxisStore[4].Axis[7].Pos17.Speed := 0;
   AxisStore[4].Axis[7].Pos17.Reached := FALSE;
   AxisStore[4].Axis[7].Pos18.Position := 0.0;
   AxisStore[4].Axis[7].Pos18.Speed := 0;
   AxisStore[4].Axis[7].Pos18.Reached := FALSE;
   AxisStore[4].Axis[7].Pos19.Position := 0.0;
   AxisStore[4].Axis[7].Pos19.Speed := 0;
   AxisStore[4].Axis[7].Pos19.Reached := FALSE;
   AxisStore[4].Axis[7].Pos20.Position := 0.0;
   AxisStore[4].Axis[7].Pos20.Speed := 0;
   AxisStore[4].Axis[7].Pos20.Reached := FALSE;
   AxisStore[4].Axis[7].Pos21.Position := 0.0;
   AxisStore[4].Axis[7].Pos21.Speed := 0;
   AxisStore[4].Axis[7].Pos21.Reached := FALSE;
   AxisStore[4].Axis[7].Pos22.Position := 0.0;
   AxisStore[4].Axis[7].Pos22.Speed := 0;
   AxisStore[4].Axis[7].Pos22.Reached := FALSE;
   AxisStore[4].Axis[7].Pos23.Position := 0.0;
   AxisStore[4].Axis[7].Pos23.Speed := 0;
   AxisStore[4].Axis[7].Pos23.Reached := FALSE;
   AxisStore[4].Axis[7].Pos24.Position := 0.0;
   AxisStore[4].Axis[7].Pos24.Speed := 0;
   AxisStore[4].Axis[7].Pos24.Reached := FALSE;
   AxisStore[4].Axis[7].Pos25.Position := 0.0;
   AxisStore[4].Axis[7].Pos25.Speed := 0;
   AxisStore[4].Axis[7].Pos25.Reached := FALSE;
   AxisStore[4].Axis[7].Pos26.Position := 0.0;
   AxisStore[4].Axis[7].Pos26.Speed := 0;
   AxisStore[4].Axis[7].Pos26.Reached := FALSE;
   AxisStore[4].Axis[7].Pos27.Position := 0.0;
   AxisStore[4].Axis[7].Pos27.Speed := 0;
   AxisStore[4].Axis[7].Pos27.Reached := FALSE;
   AxisStore[4].Axis[7].Pos28.Position := 0.0;
   AxisStore[4].Axis[7].Pos28.Speed := 0;
   AxisStore[4].Axis[7].Pos28.Reached := FALSE;
   AxisStore[4].Axis[7].Pos29.Position := 0.0;
   AxisStore[4].Axis[7].Pos29.Speed := 0;
   AxisStore[4].Axis[7].Pos29.Reached := FALSE;
   AxisStore[4].Axis[7].Pos30.Position := 0.0;
   AxisStore[4].Axis[7].Pos30.Speed := 0;
   AxisStore[4].Axis[7].Pos30.Reached := FALSE;
   AxisStore[4].Axis[8].Pos1.Position := 0.0;
   AxisStore[4].Axis[8].Pos1.Speed := 0;
   AxisStore[4].Axis[8].Pos1.Reached := FALSE;
   AxisStore[4].Axis[8].Pos2.Position := 0.0;
   AxisStore[4].Axis[8].Pos2.Speed := 0;
   AxisStore[4].Axis[8].Pos2.Reached := FALSE;
   AxisStore[4].Axis[8].Pos3.Position := 0.0;
   AxisStore[4].Axis[8].Pos3.Speed := 0;
   AxisStore[4].Axis[8].Pos3.Reached := FALSE;
   AxisStore[4].Axis[8].Pos4.Position := 0.0;
   AxisStore[4].Axis[8].Pos4.Speed := 0;
   AxisStore[4].Axis[8].Pos4.Reached := FALSE;
   AxisStore[4].Axis[8].Pos5.Position := 0.0;
   AxisStore[4].Axis[8].Pos5.Speed := 0;
   AxisStore[4].Axis[8].Pos5.Reached := FALSE;
   AxisStore[4].Axis[8].Pos6.Position := 0.0;
   AxisStore[4].Axis[8].Pos6.Speed := 0;
   AxisStore[4].Axis[8].Pos6.Reached := FALSE;
   AxisStore[4].Axis[8].Pos7.Position := 0.0;
   AxisStore[4].Axis[8].Pos7.Speed := 0;
   AxisStore[4].Axis[8].Pos7.Reached := FALSE;
   AxisStore[4].Axis[8].Pos8.Position := 0.0;
   AxisStore[4].Axis[8].Pos8.Speed := 0;
   AxisStore[4].Axis[8].Pos8.Reached := FALSE;
   AxisStore[4].Axis[8].Pos9.Position := 0.0;
   AxisStore[4].Axis[8].Pos9.Speed := 0;
   AxisStore[4].Axis[8].Pos9.Reached := FALSE;
   AxisStore[4].Axis[8].Pos10.Position := 0.0;
   AxisStore[4].Axis[8].Pos10.Speed := 0;
   AxisStore[4].Axis[8].Pos10.Reached := FALSE;
   AxisStore[4].Axis[8].Pos11.Position := 0.0;
   AxisStore[4].Axis[8].Pos11.Speed := 0;
   AxisStore[4].Axis[8].Pos11.Reached := FALSE;
   AxisStore[4].Axis[8].Pos12.Position := 0.0;
   AxisStore[4].Axis[8].Pos12.Speed := 0;
   AxisStore[4].Axis[8].Pos12.Reached := FALSE;
   AxisStore[4].Axis[8].Pos13.Position := 0.0;
   AxisStore[4].Axis[8].Pos13.Speed := 0;
   AxisStore[4].Axis[8].Pos13.Reached := FALSE;
   AxisStore[4].Axis[8].Pos14.Position := 0.0;
   AxisStore[4].Axis[8].Pos14.Speed := 0;
   AxisStore[4].Axis[8].Pos14.Reached := FALSE;
   AxisStore[4].Axis[8].Pos15.Position := 0.0;
   AxisStore[4].Axis[8].Pos15.Speed := 0;
   AxisStore[4].Axis[8].Pos15.Reached := FALSE;
   AxisStore[4].Axis[8].Pos16.Position := 0.0;
   AxisStore[4].Axis[8].Pos16.Speed := 0;
   AxisStore[4].Axis[8].Pos16.Reached := FALSE;
   AxisStore[4].Axis[8].Pos17.Position := 0.0;
   AxisStore[4].Axis[8].Pos17.Speed := 0;
   AxisStore[4].Axis[8].Pos17.Reached := FALSE;
   AxisStore[4].Axis[8].Pos18.Position := 0.0;
   AxisStore[4].Axis[8].Pos18.Speed := 0;
   AxisStore[4].Axis[8].Pos18.Reached := FALSE;
   AxisStore[4].Axis[8].Pos19.Position := 0.0;
   AxisStore[4].Axis[8].Pos19.Speed := 0;
   AxisStore[4].Axis[8].Pos19.Reached := FALSE;
   AxisStore[4].Axis[8].Pos20.Position := 0.0;
   AxisStore[4].Axis[8].Pos20.Speed := 0;
   AxisStore[4].Axis[8].Pos20.Reached := FALSE;
   AxisStore[4].Axis[8].Pos21.Position := 0.0;
   AxisStore[4].Axis[8].Pos21.Speed := 0;
   AxisStore[4].Axis[8].Pos21.Reached := FALSE;
   AxisStore[4].Axis[8].Pos22.Position := 0.0;
   AxisStore[4].Axis[8].Pos22.Speed := 0;
   AxisStore[4].Axis[8].Pos22.Reached := FALSE;
   AxisStore[4].Axis[8].Pos23.Position := 0.0;
   AxisStore[4].Axis[8].Pos23.Speed := 0;
   AxisStore[4].Axis[8].Pos23.Reached := FALSE;
   AxisStore[4].Axis[8].Pos24.Position := 0.0;
   AxisStore[4].Axis[8].Pos24.Speed := 0;
   AxisStore[4].Axis[8].Pos24.Reached := FALSE;
   AxisStore[4].Axis[8].Pos25.Position := 0.0;
   AxisStore[4].Axis[8].Pos25.Speed := 0;
   AxisStore[4].Axis[8].Pos25.Reached := FALSE;
   AxisStore[4].Axis[8].Pos26.Position := 0.0;
   AxisStore[4].Axis[8].Pos26.Speed := 0;
   AxisStore[4].Axis[8].Pos26.Reached := FALSE;
   AxisStore[4].Axis[8].Pos27.Position := 0.0;
   AxisStore[4].Axis[8].Pos27.Speed := 0;
   AxisStore[4].Axis[8].Pos27.Reached := FALSE;
   AxisStore[4].Axis[8].Pos28.Position := 0.0;
   AxisStore[4].Axis[8].Pos28.Speed := 0;
   AxisStore[4].Axis[8].Pos28.Reached := FALSE;
   AxisStore[4].Axis[8].Pos29.Position := 0.0;
   AxisStore[4].Axis[8].Pos29.Speed := 0;
   AxisStore[4].Axis[8].Pos29.Reached := FALSE;
   AxisStore[4].Axis[8].Pos30.Position := 0.0;
   AxisStore[4].Axis[8].Pos30.Speed := 0;
   AxisStore[4].Axis[8].Pos30.Reached := FALSE;
   AxisStore[4].Axis[9].Pos1.Position := 0.0;
   AxisStore[4].Axis[9].Pos1.Speed := 0;
   AxisStore[4].Axis[9].Pos1.Reached := FALSE;
   AxisStore[4].Axis[9].Pos2.Position := 0.0;
   AxisStore[4].Axis[9].Pos2.Speed := 0;
   AxisStore[4].Axis[9].Pos2.Reached := FALSE;
   AxisStore[4].Axis[9].Pos3.Position := 0.0;
   AxisStore[4].Axis[9].Pos3.Speed := 0;
   AxisStore[4].Axis[9].Pos3.Reached := FALSE;
   AxisStore[4].Axis[9].Pos4.Position := 0.0;
   AxisStore[4].Axis[9].Pos4.Speed := 0;
   AxisStore[4].Axis[9].Pos4.Reached := FALSE;
   AxisStore[4].Axis[9].Pos5.Position := 0.0;
   AxisStore[4].Axis[9].Pos5.Speed := 0;
   AxisStore[4].Axis[9].Pos5.Reached := FALSE;
   AxisStore[4].Axis[9].Pos6.Position := 0.0;
   AxisStore[4].Axis[9].Pos6.Speed := 0;
   AxisStore[4].Axis[9].Pos6.Reached := FALSE;
   AxisStore[4].Axis[9].Pos7.Position := 0.0;
   AxisStore[4].Axis[9].Pos7.Speed := 0;
   AxisStore[4].Axis[9].Pos7.Reached := FALSE;
   AxisStore[4].Axis[9].Pos8.Position := 0.0;
   AxisStore[4].Axis[9].Pos8.Speed := 0;
   AxisStore[4].Axis[9].Pos8.Reached := FALSE;
   AxisStore[4].Axis[9].Pos9.Position := 0.0;
   AxisStore[4].Axis[9].Pos9.Speed := 0;
   AxisStore[4].Axis[9].Pos9.Reached := FALSE;
   AxisStore[4].Axis[9].Pos10.Position := 0.0;
   AxisStore[4].Axis[9].Pos10.Speed := 0;
   AxisStore[4].Axis[9].Pos10.Reached := FALSE;
   AxisStore[4].Axis[9].Pos11.Position := 0.0;
   AxisStore[4].Axis[9].Pos11.Speed := 0;
   AxisStore[4].Axis[9].Pos11.Reached := FALSE;
   AxisStore[4].Axis[9].Pos12.Position := 0.0;
   AxisStore[4].Axis[9].Pos12.Speed := 0;
   AxisStore[4].Axis[9].Pos12.Reached := FALSE;
   AxisStore[4].Axis[9].Pos13.Position := 0.0;
   AxisStore[4].Axis[9].Pos13.Speed := 0;
   AxisStore[4].Axis[9].Pos13.Reached := FALSE;
   AxisStore[4].Axis[9].Pos14.Position := 0.0;
   AxisStore[4].Axis[9].Pos14.Speed := 0;
   AxisStore[4].Axis[9].Pos14.Reached := FALSE;
   AxisStore[4].Axis[9].Pos15.Position := 0.0;
   AxisStore[4].Axis[9].Pos15.Speed := 0;
   AxisStore[4].Axis[9].Pos15.Reached := FALSE;
   AxisStore[4].Axis[9].Pos16.Position := 0.0;
   AxisStore[4].Axis[9].Pos16.Speed := 0;
   AxisStore[4].Axis[9].Pos16.Reached := FALSE;
   AxisStore[4].Axis[9].Pos17.Position := 0.0;
   AxisStore[4].Axis[9].Pos17.Speed := 0;
   AxisStore[4].Axis[9].Pos17.Reached := FALSE;
   AxisStore[4].Axis[9].Pos18.Position := 0.0;
   AxisStore[4].Axis[9].Pos18.Speed := 0;
   AxisStore[4].Axis[9].Pos18.Reached := FALSE;
   AxisStore[4].Axis[9].Pos19.Position := 0.0;
   AxisStore[4].Axis[9].Pos19.Speed := 0;
   AxisStore[4].Axis[9].Pos19.Reached := FALSE;
   AxisStore[4].Axis[9].Pos20.Position := 0.0;
   AxisStore[4].Axis[9].Pos20.Speed := 0;
   AxisStore[4].Axis[9].Pos20.Reached := FALSE;
   AxisStore[4].Axis[9].Pos21.Position := 0.0;
   AxisStore[4].Axis[9].Pos21.Speed := 0;
   AxisStore[4].Axis[9].Pos21.Reached := FALSE;
   AxisStore[4].Axis[9].Pos22.Position := 0.0;
   AxisStore[4].Axis[9].Pos22.Speed := 0;
   AxisStore[4].Axis[9].Pos22.Reached := FALSE;
   AxisStore[4].Axis[9].Pos23.Position := 0.0;
   AxisStore[4].Axis[9].Pos23.Speed := 0;
   AxisStore[4].Axis[9].Pos23.Reached := FALSE;
   AxisStore[4].Axis[9].Pos24.Position := 0.0;
   AxisStore[4].Axis[9].Pos24.Speed := 0;
   AxisStore[4].Axis[9].Pos24.Reached := FALSE;
   AxisStore[4].Axis[9].Pos25.Position := 0.0;
   AxisStore[4].Axis[9].Pos25.Speed := 0;
   AxisStore[4].Axis[9].Pos25.Reached := FALSE;
   AxisStore[4].Axis[9].Pos26.Position := 0.0;
   AxisStore[4].Axis[9].Pos26.Speed := 0;
   AxisStore[4].Axis[9].Pos26.Reached := FALSE;
   AxisStore[4].Axis[9].Pos27.Position := 0.0;
   AxisStore[4].Axis[9].Pos27.Speed := 0;
   AxisStore[4].Axis[9].Pos27.Reached := FALSE;
   AxisStore[4].Axis[9].Pos28.Position := 0.0;
   AxisStore[4].Axis[9].Pos28.Speed := 0;
   AxisStore[4].Axis[9].Pos28.Reached := FALSE;
   AxisStore[4].Axis[9].Pos29.Position := 0.0;
   AxisStore[4].Axis[9].Pos29.Speed := 0;
   AxisStore[4].Axis[9].Pos29.Reached := FALSE;
   AxisStore[4].Axis[9].Pos30.Position := 0.0;
   AxisStore[4].Axis[9].Pos30.Speed := 0;
   AxisStore[4].Axis[9].Pos30.Reached := FALSE;
   AxisStore[4].Axis[10].Pos1.Position := 0.0;
   AxisStore[4].Axis[10].Pos1.Speed := 0;
   AxisStore[4].Axis[10].Pos1.Reached := FALSE;
   AxisStore[4].Axis[10].Pos2.Position := 0.0;
   AxisStore[4].Axis[10].Pos2.Speed := 0;
   AxisStore[4].Axis[10].Pos2.Reached := FALSE;
   AxisStore[4].Axis[10].Pos3.Position := 0.0;
   AxisStore[4].Axis[10].Pos3.Speed := 0;
   AxisStore[4].Axis[10].Pos3.Reached := FALSE;
   AxisStore[4].Axis[10].Pos4.Position := 0.0;
   AxisStore[4].Axis[10].Pos4.Speed := 0;
   AxisStore[4].Axis[10].Pos4.Reached := FALSE;
   AxisStore[4].Axis[10].Pos5.Position := 0.0;
   AxisStore[4].Axis[10].Pos5.Speed := 0;
   AxisStore[4].Axis[10].Pos5.Reached := FALSE;
   AxisStore[4].Axis[10].Pos6.Position := 0.0;
   AxisStore[4].Axis[10].Pos6.Speed := 0;
   AxisStore[4].Axis[10].Pos6.Reached := FALSE;
   AxisStore[4].Axis[10].Pos7.Position := 0.0;
   AxisStore[4].Axis[10].Pos7.Speed := 0;
   AxisStore[4].Axis[10].Pos7.Reached := FALSE;
   AxisStore[4].Axis[10].Pos8.Position := 0.0;
   AxisStore[4].Axis[10].Pos8.Speed := 0;
   AxisStore[4].Axis[10].Pos8.Reached := FALSE;
   AxisStore[4].Axis[10].Pos9.Position := 0.0;
   AxisStore[4].Axis[10].Pos9.Speed := 0;
   AxisStore[4].Axis[10].Pos9.Reached := FALSE;
   AxisStore[4].Axis[10].Pos10.Position := 0.0;
   AxisStore[4].Axis[10].Pos10.Speed := 0;
   AxisStore[4].Axis[10].Pos10.Reached := FALSE;
   AxisStore[4].Axis[10].Pos11.Position := 0.0;
   AxisStore[4].Axis[10].Pos11.Speed := 0;
   AxisStore[4].Axis[10].Pos11.Reached := FALSE;
   AxisStore[4].Axis[10].Pos12.Position := 0.0;
   AxisStore[4].Axis[10].Pos12.Speed := 0;
   AxisStore[4].Axis[10].Pos12.Reached := FALSE;
   AxisStore[4].Axis[10].Pos13.Position := 0.0;
   AxisStore[4].Axis[10].Pos13.Speed := 0;
   AxisStore[4].Axis[10].Pos13.Reached := FALSE;
   AxisStore[4].Axis[10].Pos14.Position := 0.0;
   AxisStore[4].Axis[10].Pos14.Speed := 0;
   AxisStore[4].Axis[10].Pos14.Reached := FALSE;
   AxisStore[4].Axis[10].Pos15.Position := 0.0;
   AxisStore[4].Axis[10].Pos15.Speed := 0;
   AxisStore[4].Axis[10].Pos15.Reached := FALSE;
   AxisStore[4].Axis[10].Pos16.Position := 0.0;
   AxisStore[4].Axis[10].Pos16.Speed := 0;
   AxisStore[4].Axis[10].Pos16.Reached := FALSE;
   AxisStore[4].Axis[10].Pos17.Position := 0.0;
   AxisStore[4].Axis[10].Pos17.Speed := 0;
   AxisStore[4].Axis[10].Pos17.Reached := FALSE;
   AxisStore[4].Axis[10].Pos18.Position := 0.0;
   AxisStore[4].Axis[10].Pos18.Speed := 0;
   AxisStore[4].Axis[10].Pos18.Reached := FALSE;
   AxisStore[4].Axis[10].Pos19.Position := 0.0;
   AxisStore[4].Axis[10].Pos19.Speed := 0;
   AxisStore[4].Axis[10].Pos19.Reached := FALSE;
   AxisStore[4].Axis[10].Pos20.Position := 0.0;
   AxisStore[4].Axis[10].Pos20.Speed := 0;
   AxisStore[4].Axis[10].Pos20.Reached := FALSE;
   AxisStore[4].Axis[10].Pos21.Position := 0.0;
   AxisStore[4].Axis[10].Pos21.Speed := 0;
   AxisStore[4].Axis[10].Pos21.Reached := FALSE;
   AxisStore[4].Axis[10].Pos22.Position := 0.0;
   AxisStore[4].Axis[10].Pos22.Speed := 0;
   AxisStore[4].Axis[10].Pos22.Reached := FALSE;
   AxisStore[4].Axis[10].Pos23.Position := 0.0;
   AxisStore[4].Axis[10].Pos23.Speed := 0;
   AxisStore[4].Axis[10].Pos23.Reached := FALSE;
   AxisStore[4].Axis[10].Pos24.Position := 0.0;
   AxisStore[4].Axis[10].Pos24.Speed := 0;
   AxisStore[4].Axis[10].Pos24.Reached := FALSE;
   AxisStore[4].Axis[10].Pos25.Position := 0.0;
   AxisStore[4].Axis[10].Pos25.Speed := 0;
   AxisStore[4].Axis[10].Pos25.Reached := FALSE;
   AxisStore[4].Axis[10].Pos26.Position := 0.0;
   AxisStore[4].Axis[10].Pos26.Speed := 0;
   AxisStore[4].Axis[10].Pos26.Reached := FALSE;
   AxisStore[4].Axis[10].Pos27.Position := 0.0;
   AxisStore[4].Axis[10].Pos27.Speed := 0;
   AxisStore[4].Axis[10].Pos27.Reached := FALSE;
   AxisStore[4].Axis[10].Pos28.Position := 0.0;
   AxisStore[4].Axis[10].Pos28.Speed := 0;
   AxisStore[4].Axis[10].Pos28.Reached := FALSE;
   AxisStore[4].Axis[10].Pos29.Position := 0.0;
   AxisStore[4].Axis[10].Pos29.Speed := 0;
   AxisStore[4].Axis[10].Pos29.Reached := FALSE;
   AxisStore[4].Axis[10].Pos30.Position := 0.0;
   AxisStore[4].Axis[10].Pos30.Speed := 0;
   AxisStore[4].Axis[10].Pos30.Reached := FALSE;
   AxisStore[4].Axis[11].Pos1.Position := 0.0;
   AxisStore[4].Axis[11].Pos1.Speed := 0;
   AxisStore[4].Axis[11].Pos1.Reached := FALSE;
   AxisStore[4].Axis[11].Pos2.Position := 0.0;
   AxisStore[4].Axis[11].Pos2.Speed := 0;
   AxisStore[4].Axis[11].Pos2.Reached := FALSE;
   AxisStore[4].Axis[11].Pos3.Position := 0.0;
   AxisStore[4].Axis[11].Pos3.Speed := 0;
   AxisStore[4].Axis[11].Pos3.Reached := FALSE;
   AxisStore[4].Axis[11].Pos4.Position := 0.0;
   AxisStore[4].Axis[11].Pos4.Speed := 0;
   AxisStore[4].Axis[11].Pos4.Reached := FALSE;
   AxisStore[4].Axis[11].Pos5.Position := 0.0;
   AxisStore[4].Axis[11].Pos5.Speed := 0;
   AxisStore[4].Axis[11].Pos5.Reached := FALSE;
   AxisStore[4].Axis[11].Pos6.Position := 0.0;
   AxisStore[4].Axis[11].Pos6.Speed := 0;
   AxisStore[4].Axis[11].Pos6.Reached := FALSE;
   AxisStore[4].Axis[11].Pos7.Position := 0.0;
   AxisStore[4].Axis[11].Pos7.Speed := 0;
   AxisStore[4].Axis[11].Pos7.Reached := FALSE;
   AxisStore[4].Axis[11].Pos8.Position := 0.0;
   AxisStore[4].Axis[11].Pos8.Speed := 0;
   AxisStore[4].Axis[11].Pos8.Reached := FALSE;
   AxisStore[4].Axis[11].Pos9.Position := 0.0;
   AxisStore[4].Axis[11].Pos9.Speed := 0;
   AxisStore[4].Axis[11].Pos9.Reached := FALSE;
   AxisStore[4].Axis[11].Pos10.Position := 0.0;
   AxisStore[4].Axis[11].Pos10.Speed := 0;
   AxisStore[4].Axis[11].Pos10.Reached := FALSE;
   AxisStore[4].Axis[11].Pos11.Position := 0.0;
   AxisStore[4].Axis[11].Pos11.Speed := 0;
   AxisStore[4].Axis[11].Pos11.Reached := FALSE;
   AxisStore[4].Axis[11].Pos12.Position := 0.0;
   AxisStore[4].Axis[11].Pos12.Speed := 0;
   AxisStore[4].Axis[11].Pos12.Reached := FALSE;
   AxisStore[4].Axis[11].Pos13.Position := 0.0;
   AxisStore[4].Axis[11].Pos13.Speed := 0;
   AxisStore[4].Axis[11].Pos13.Reached := FALSE;
   AxisStore[4].Axis[11].Pos14.Position := 0.0;
   AxisStore[4].Axis[11].Pos14.Speed := 0;
   AxisStore[4].Axis[11].Pos14.Reached := FALSE;
   AxisStore[4].Axis[11].Pos15.Position := 0.0;
   AxisStore[4].Axis[11].Pos15.Speed := 0;
   AxisStore[4].Axis[11].Pos15.Reached := FALSE;
   AxisStore[4].Axis[11].Pos16.Position := 0.0;
   AxisStore[4].Axis[11].Pos16.Speed := 0;
   AxisStore[4].Axis[11].Pos16.Reached := FALSE;
   AxisStore[4].Axis[11].Pos17.Position := 0.0;
   AxisStore[4].Axis[11].Pos17.Speed := 0;
   AxisStore[4].Axis[11].Pos17.Reached := FALSE;
   AxisStore[4].Axis[11].Pos18.Position := 0.0;
   AxisStore[4].Axis[11].Pos18.Speed := 0;
   AxisStore[4].Axis[11].Pos18.Reached := FALSE;
   AxisStore[4].Axis[11].Pos19.Position := 0.0;
   AxisStore[4].Axis[11].Pos19.Speed := 0;
   AxisStore[4].Axis[11].Pos19.Reached := FALSE;
   AxisStore[4].Axis[11].Pos20.Position := 0.0;
   AxisStore[4].Axis[11].Pos20.Speed := 0;
   AxisStore[4].Axis[11].Pos20.Reached := FALSE;
   AxisStore[4].Axis[11].Pos21.Position := 0.0;
   AxisStore[4].Axis[11].Pos21.Speed := 0;
   AxisStore[4].Axis[11].Pos21.Reached := FALSE;
   AxisStore[4].Axis[11].Pos22.Position := 0.0;
   AxisStore[4].Axis[11].Pos22.Speed := 0;
   AxisStore[4].Axis[11].Pos22.Reached := FALSE;
   AxisStore[4].Axis[11].Pos23.Position := 0.0;
   AxisStore[4].Axis[11].Pos23.Speed := 0;
   AxisStore[4].Axis[11].Pos23.Reached := FALSE;
   AxisStore[4].Axis[11].Pos24.Position := 0.0;
   AxisStore[4].Axis[11].Pos24.Speed := 0;
   AxisStore[4].Axis[11].Pos24.Reached := FALSE;
   AxisStore[4].Axis[11].Pos25.Position := 0.0;
   AxisStore[4].Axis[11].Pos25.Speed := 0;
   AxisStore[4].Axis[11].Pos25.Reached := FALSE;
   AxisStore[4].Axis[11].Pos26.Position := 0.0;
   AxisStore[4].Axis[11].Pos26.Speed := 0;
   AxisStore[4].Axis[11].Pos26.Reached := FALSE;
   AxisStore[4].Axis[11].Pos27.Position := 0.0;
   AxisStore[4].Axis[11].Pos27.Speed := 0;
   AxisStore[4].Axis[11].Pos27.Reached := FALSE;
   AxisStore[4].Axis[11].Pos28.Position := 0.0;
   AxisStore[4].Axis[11].Pos28.Speed := 0;
   AxisStore[4].Axis[11].Pos28.Reached := FALSE;
   AxisStore[4].Axis[11].Pos29.Position := 0.0;
   AxisStore[4].Axis[11].Pos29.Speed := 0;
   AxisStore[4].Axis[11].Pos29.Reached := FALSE;
   AxisStore[4].Axis[11].Pos30.Position := 0.0;
   AxisStore[4].Axis[11].Pos30.Speed := 0;
   AxisStore[4].Axis[11].Pos30.Reached := FALSE;
   AxisStore[4].Axis[12].Pos1.Position := 0.0;
   AxisStore[4].Axis[12].Pos1.Speed := 0;
   AxisStore[4].Axis[12].Pos1.Reached := FALSE;
   AxisStore[4].Axis[12].Pos2.Position := 0.0;
   AxisStore[4].Axis[12].Pos2.Speed := 0;
   AxisStore[4].Axis[12].Pos2.Reached := FALSE;
   AxisStore[4].Axis[12].Pos3.Position := 0.0;
   AxisStore[4].Axis[12].Pos3.Speed := 0;
   AxisStore[4].Axis[12].Pos3.Reached := FALSE;
   AxisStore[4].Axis[12].Pos4.Position := 0.0;
   AxisStore[4].Axis[12].Pos4.Speed := 0;
   AxisStore[4].Axis[12].Pos4.Reached := FALSE;
   AxisStore[4].Axis[12].Pos5.Position := 0.0;
   AxisStore[4].Axis[12].Pos5.Speed := 0;
   AxisStore[4].Axis[12].Pos5.Reached := FALSE;
   AxisStore[4].Axis[12].Pos6.Position := 0.0;
   AxisStore[4].Axis[12].Pos6.Speed := 0;
   AxisStore[4].Axis[12].Pos6.Reached := FALSE;
   AxisStore[4].Axis[12].Pos7.Position := 0.0;
   AxisStore[4].Axis[12].Pos7.Speed := 0;
   AxisStore[4].Axis[12].Pos7.Reached := FALSE;
   AxisStore[4].Axis[12].Pos8.Position := 0.0;
   AxisStore[4].Axis[12].Pos8.Speed := 0;
   AxisStore[4].Axis[12].Pos8.Reached := FALSE;
   AxisStore[4].Axis[12].Pos9.Position := 0.0;
   AxisStore[4].Axis[12].Pos9.Speed := 0;
   AxisStore[4].Axis[12].Pos9.Reached := FALSE;
   AxisStore[4].Axis[12].Pos10.Position := 0.0;
   AxisStore[4].Axis[12].Pos10.Speed := 0;
   AxisStore[4].Axis[12].Pos10.Reached := FALSE;
   AxisStore[4].Axis[12].Pos11.Position := 0.0;
   AxisStore[4].Axis[12].Pos11.Speed := 0;
   AxisStore[4].Axis[12].Pos11.Reached := FALSE;
   AxisStore[4].Axis[12].Pos12.Position := 0.0;
   AxisStore[4].Axis[12].Pos12.Speed := 0;
   AxisStore[4].Axis[12].Pos12.Reached := FALSE;
   AxisStore[4].Axis[12].Pos13.Position := 0.0;
   AxisStore[4].Axis[12].Pos13.Speed := 0;
   AxisStore[4].Axis[12].Pos13.Reached := FALSE;
   AxisStore[4].Axis[12].Pos14.Position := 0.0;
   AxisStore[4].Axis[12].Pos14.Speed := 0;
   AxisStore[4].Axis[12].Pos14.Reached := FALSE;
   AxisStore[4].Axis[12].Pos15.Position := 0.0;
   AxisStore[4].Axis[12].Pos15.Speed := 0;
   AxisStore[4].Axis[12].Pos15.Reached := FALSE;
   AxisStore[4].Axis[12].Pos16.Position := 0.0;
   AxisStore[4].Axis[12].Pos16.Speed := 0;
   AxisStore[4].Axis[12].Pos16.Reached := FALSE;
   AxisStore[4].Axis[12].Pos17.Position := 0.0;
   AxisStore[4].Axis[12].Pos17.Speed := 0;
   AxisStore[4].Axis[12].Pos17.Reached := FALSE;
   AxisStore[4].Axis[12].Pos18.Position := 0.0;
   AxisStore[4].Axis[12].Pos18.Speed := 0;
   AxisStore[4].Axis[12].Pos18.Reached := FALSE;
   AxisStore[4].Axis[12].Pos19.Position := 0.0;
   AxisStore[4].Axis[12].Pos19.Speed := 0;
   AxisStore[4].Axis[12].Pos19.Reached := FALSE;
   AxisStore[4].Axis[12].Pos20.Position := 0.0;
   AxisStore[4].Axis[12].Pos20.Speed := 0;
   AxisStore[4].Axis[12].Pos20.Reached := FALSE;
   AxisStore[4].Axis[12].Pos21.Position := 0.0;
   AxisStore[4].Axis[12].Pos21.Speed := 0;
   AxisStore[4].Axis[12].Pos21.Reached := FALSE;
   AxisStore[4].Axis[12].Pos22.Position := 0.0;
   AxisStore[4].Axis[12].Pos22.Speed := 0;
   AxisStore[4].Axis[12].Pos22.Reached := FALSE;
   AxisStore[4].Axis[12].Pos23.Position := 0.0;
   AxisStore[4].Axis[12].Pos23.Speed := 0;
   AxisStore[4].Axis[12].Pos23.Reached := FALSE;
   AxisStore[4].Axis[12].Pos24.Position := 0.0;
   AxisStore[4].Axis[12].Pos24.Speed := 0;
   AxisStore[4].Axis[12].Pos24.Reached := FALSE;
   AxisStore[4].Axis[12].Pos25.Position := 0.0;
   AxisStore[4].Axis[12].Pos25.Speed := 0;
   AxisStore[4].Axis[12].Pos25.Reached := FALSE;
   AxisStore[4].Axis[12].Pos26.Position := 0.0;
   AxisStore[4].Axis[12].Pos26.Speed := 0;
   AxisStore[4].Axis[12].Pos26.Reached := FALSE;
   AxisStore[4].Axis[12].Pos27.Position := 0.0;
   AxisStore[4].Axis[12].Pos27.Speed := 0;
   AxisStore[4].Axis[12].Pos27.Reached := FALSE;
   AxisStore[4].Axis[12].Pos28.Position := 0.0;
   AxisStore[4].Axis[12].Pos28.Speed := 0;
   AxisStore[4].Axis[12].Pos28.Reached := FALSE;
   AxisStore[4].Axis[12].Pos29.Position := 0.0;
   AxisStore[4].Axis[12].Pos29.Speed := 0;
   AxisStore[4].Axis[12].Pos29.Reached := FALSE;
   AxisStore[4].Axis[12].Pos30.Position := 0.0;
   AxisStore[4].Axis[12].Pos30.Speed := 0;
   AxisStore[4].Axis[12].Pos30.Reached := FALSE;
   AxisStore[4].Axis[13].Pos1.Position := 0.0;
   AxisStore[4].Axis[13].Pos1.Speed := 0;
   AxisStore[4].Axis[13].Pos1.Reached := FALSE;
   AxisStore[4].Axis[13].Pos2.Position := 0.0;
   AxisStore[4].Axis[13].Pos2.Speed := 0;
   AxisStore[4].Axis[13].Pos2.Reached := FALSE;
   AxisStore[4].Axis[13].Pos3.Position := 0.0;
   AxisStore[4].Axis[13].Pos3.Speed := 0;
   AxisStore[4].Axis[13].Pos3.Reached := FALSE;
   AxisStore[4].Axis[13].Pos4.Position := 0.0;
   AxisStore[4].Axis[13].Pos4.Speed := 0;
   AxisStore[4].Axis[13].Pos4.Reached := FALSE;
   AxisStore[4].Axis[13].Pos5.Position := 0.0;
   AxisStore[4].Axis[13].Pos5.Speed := 0;
   AxisStore[4].Axis[13].Pos5.Reached := FALSE;
   AxisStore[4].Axis[13].Pos6.Position := 0.0;
   AxisStore[4].Axis[13].Pos6.Speed := 0;
   AxisStore[4].Axis[13].Pos6.Reached := FALSE;
   AxisStore[4].Axis[13].Pos7.Position := 0.0;
   AxisStore[4].Axis[13].Pos7.Speed := 0;
   AxisStore[4].Axis[13].Pos7.Reached := FALSE;
   AxisStore[4].Axis[13].Pos8.Position := 0.0;
   AxisStore[4].Axis[13].Pos8.Speed := 0;
   AxisStore[4].Axis[13].Pos8.Reached := FALSE;
   AxisStore[4].Axis[13].Pos9.Position := 0.0;
   AxisStore[4].Axis[13].Pos9.Speed := 0;
   AxisStore[4].Axis[13].Pos9.Reached := FALSE;
   AxisStore[4].Axis[13].Pos10.Position := 0.0;
   AxisStore[4].Axis[13].Pos10.Speed := 0;
   AxisStore[4].Axis[13].Pos10.Reached := FALSE;
   AxisStore[4].Axis[13].Pos11.Position := 0.0;
   AxisStore[4].Axis[13].Pos11.Speed := 0;
   AxisStore[4].Axis[13].Pos11.Reached := FALSE;
   AxisStore[4].Axis[13].Pos12.Position := 0.0;
   AxisStore[4].Axis[13].Pos12.Speed := 0;
   AxisStore[4].Axis[13].Pos12.Reached := FALSE;
   AxisStore[4].Axis[13].Pos13.Position := 0.0;
   AxisStore[4].Axis[13].Pos13.Speed := 0;
   AxisStore[4].Axis[13].Pos13.Reached := FALSE;
   AxisStore[4].Axis[13].Pos14.Position := 0.0;
   AxisStore[4].Axis[13].Pos14.Speed := 0;
   AxisStore[4].Axis[13].Pos14.Reached := FALSE;
   AxisStore[4].Axis[13].Pos15.Position := 0.0;
   AxisStore[4].Axis[13].Pos15.Speed := 0;
   AxisStore[4].Axis[13].Pos15.Reached := FALSE;
   AxisStore[4].Axis[13].Pos16.Position := 0.0;
   AxisStore[4].Axis[13].Pos16.Speed := 0;
   AxisStore[4].Axis[13].Pos16.Reached := FALSE;
   AxisStore[4].Axis[13].Pos17.Position := 0.0;
   AxisStore[4].Axis[13].Pos17.Speed := 0;
   AxisStore[4].Axis[13].Pos17.Reached := FALSE;
   AxisStore[4].Axis[13].Pos18.Position := 0.0;
   AxisStore[4].Axis[13].Pos18.Speed := 0;
   AxisStore[4].Axis[13].Pos18.Reached := FALSE;
   AxisStore[4].Axis[13].Pos19.Position := 0.0;
   AxisStore[4].Axis[13].Pos19.Speed := 0;
   AxisStore[4].Axis[13].Pos19.Reached := FALSE;
   AxisStore[4].Axis[13].Pos20.Position := 0.0;
   AxisStore[4].Axis[13].Pos20.Speed := 0;
   AxisStore[4].Axis[13].Pos20.Reached := FALSE;
   AxisStore[4].Axis[13].Pos21.Position := 0.0;
   AxisStore[4].Axis[13].Pos21.Speed := 0;
   AxisStore[4].Axis[13].Pos21.Reached := FALSE;
   AxisStore[4].Axis[13].Pos22.Position := 0.0;
   AxisStore[4].Axis[13].Pos22.Speed := 0;
   AxisStore[4].Axis[13].Pos22.Reached := FALSE;
   AxisStore[4].Axis[13].Pos23.Position := 0.0;
   AxisStore[4].Axis[13].Pos23.Speed := 0;
   AxisStore[4].Axis[13].Pos23.Reached := FALSE;
   AxisStore[4].Axis[13].Pos24.Position := 0.0;
   AxisStore[4].Axis[13].Pos24.Speed := 0;
   AxisStore[4].Axis[13].Pos24.Reached := FALSE;
   AxisStore[4].Axis[13].Pos25.Position := 0.0;
   AxisStore[4].Axis[13].Pos25.Speed := 0;
   AxisStore[4].Axis[13].Pos25.Reached := FALSE;
   AxisStore[4].Axis[13].Pos26.Position := 0.0;
   AxisStore[4].Axis[13].Pos26.Speed := 0;
   AxisStore[4].Axis[13].Pos26.Reached := FALSE;
   AxisStore[4].Axis[13].Pos27.Position := 0.0;
   AxisStore[4].Axis[13].Pos27.Speed := 0;
   AxisStore[4].Axis[13].Pos27.Reached := FALSE;
   AxisStore[4].Axis[13].Pos28.Position := 0.0;
   AxisStore[4].Axis[13].Pos28.Speed := 0;
   AxisStore[4].Axis[13].Pos28.Reached := FALSE;
   AxisStore[4].Axis[13].Pos29.Position := 0.0;
   AxisStore[4].Axis[13].Pos29.Speed := 0;
   AxisStore[4].Axis[13].Pos29.Reached := FALSE;
   AxisStore[4].Axis[13].Pos30.Position := 0.0;
   AxisStore[4].Axis[13].Pos30.Speed := 0;
   AxisStore[4].Axis[13].Pos30.Reached := FALSE;
   AxisStore[4].Axis[14].Pos1.Position := 0.0;
   AxisStore[4].Axis[14].Pos1.Speed := 0;
   AxisStore[4].Axis[14].Pos1.Reached := FALSE;
   AxisStore[4].Axis[14].Pos2.Position := 0.0;
   AxisStore[4].Axis[14].Pos2.Speed := 0;
   AxisStore[4].Axis[14].Pos2.Reached := FALSE;
   AxisStore[4].Axis[14].Pos3.Position := 0.0;
   AxisStore[4].Axis[14].Pos3.Speed := 0;
   AxisStore[4].Axis[14].Pos3.Reached := FALSE;
   AxisStore[4].Axis[14].Pos4.Position := 0.0;
   AxisStore[4].Axis[14].Pos4.Speed := 0;
   AxisStore[4].Axis[14].Pos4.Reached := FALSE;
   AxisStore[4].Axis[14].Pos5.Position := 0.0;
   AxisStore[4].Axis[14].Pos5.Speed := 0;
   AxisStore[4].Axis[14].Pos5.Reached := FALSE;
   AxisStore[4].Axis[14].Pos6.Position := 0.0;
   AxisStore[4].Axis[14].Pos6.Speed := 0;
   AxisStore[4].Axis[14].Pos6.Reached := FALSE;
   AxisStore[4].Axis[14].Pos7.Position := 0.0;
   AxisStore[4].Axis[14].Pos7.Speed := 0;
   AxisStore[4].Axis[14].Pos7.Reached := FALSE;
   AxisStore[4].Axis[14].Pos8.Position := 0.0;
   AxisStore[4].Axis[14].Pos8.Speed := 0;
   AxisStore[4].Axis[14].Pos8.Reached := FALSE;
   AxisStore[4].Axis[14].Pos9.Position := 0.0;
   AxisStore[4].Axis[14].Pos9.Speed := 0;
   AxisStore[4].Axis[14].Pos9.Reached := FALSE;
   AxisStore[4].Axis[14].Pos10.Position := 0.0;
   AxisStore[4].Axis[14].Pos10.Speed := 0;
   AxisStore[4].Axis[14].Pos10.Reached := FALSE;
   AxisStore[4].Axis[14].Pos11.Position := 0.0;
   AxisStore[4].Axis[14].Pos11.Speed := 0;
   AxisStore[4].Axis[14].Pos11.Reached := FALSE;
   AxisStore[4].Axis[14].Pos12.Position := 0.0;
   AxisStore[4].Axis[14].Pos12.Speed := 0;
   AxisStore[4].Axis[14].Pos12.Reached := FALSE;
   AxisStore[4].Axis[14].Pos13.Position := 0.0;
   AxisStore[4].Axis[14].Pos13.Speed := 0;
   AxisStore[4].Axis[14].Pos13.Reached := FALSE;
   AxisStore[4].Axis[14].Pos14.Position := 0.0;
   AxisStore[4].Axis[14].Pos14.Speed := 0;
   AxisStore[4].Axis[14].Pos14.Reached := FALSE;
   AxisStore[4].Axis[14].Pos15.Position := 0.0;
   AxisStore[4].Axis[14].Pos15.Speed := 0;
   AxisStore[4].Axis[14].Pos15.Reached := FALSE;
   AxisStore[4].Axis[14].Pos16.Position := 0.0;
   AxisStore[4].Axis[14].Pos16.Speed := 0;
   AxisStore[4].Axis[14].Pos16.Reached := FALSE;
   AxisStore[4].Axis[14].Pos17.Position := 0.0;
   AxisStore[4].Axis[14].Pos17.Speed := 0;
   AxisStore[4].Axis[14].Pos17.Reached := FALSE;
   AxisStore[4].Axis[14].Pos18.Position := 0.0;
   AxisStore[4].Axis[14].Pos18.Speed := 0;
   AxisStore[4].Axis[14].Pos18.Reached := FALSE;
   AxisStore[4].Axis[14].Pos19.Position := 0.0;
   AxisStore[4].Axis[14].Pos19.Speed := 0;
   AxisStore[4].Axis[14].Pos19.Reached := FALSE;
   AxisStore[4].Axis[14].Pos20.Position := 0.0;
   AxisStore[4].Axis[14].Pos20.Speed := 0;
   AxisStore[4].Axis[14].Pos20.Reached := FALSE;
   AxisStore[4].Axis[14].Pos21.Position := 0.0;
   AxisStore[4].Axis[14].Pos21.Speed := 0;
   AxisStore[4].Axis[14].Pos21.Reached := FALSE;
   AxisStore[4].Axis[14].Pos22.Position := 0.0;
   AxisStore[4].Axis[14].Pos22.Speed := 0;
   AxisStore[4].Axis[14].Pos22.Reached := FALSE;
   AxisStore[4].Axis[14].Pos23.Position := 0.0;
   AxisStore[4].Axis[14].Pos23.Speed := 0;
   AxisStore[4].Axis[14].Pos23.Reached := FALSE;
   AxisStore[4].Axis[14].Pos24.Position := 0.0;
   AxisStore[4].Axis[14].Pos24.Speed := 0;
   AxisStore[4].Axis[14].Pos24.Reached := FALSE;
   AxisStore[4].Axis[14].Pos25.Position := 0.0;
   AxisStore[4].Axis[14].Pos25.Speed := 0;
   AxisStore[4].Axis[14].Pos25.Reached := FALSE;
   AxisStore[4].Axis[14].Pos26.Position := 0.0;
   AxisStore[4].Axis[14].Pos26.Speed := 0;
   AxisStore[4].Axis[14].Pos26.Reached := FALSE;
   AxisStore[4].Axis[14].Pos27.Position := 0.0;
   AxisStore[4].Axis[14].Pos27.Speed := 0;
   AxisStore[4].Axis[14].Pos27.Reached := FALSE;
   AxisStore[4].Axis[14].Pos28.Position := 0.0;
   AxisStore[4].Axis[14].Pos28.Speed := 0;
   AxisStore[4].Axis[14].Pos28.Reached := FALSE;
   AxisStore[4].Axis[14].Pos29.Position := 0.0;
   AxisStore[4].Axis[14].Pos29.Speed := 0;
   AxisStore[4].Axis[14].Pos29.Reached := FALSE;
   AxisStore[4].Axis[14].Pos30.Position := 0.0;
   AxisStore[4].Axis[14].Pos30.Speed := 0;
   AxisStore[4].Axis[14].Pos30.Reached := FALSE;
   AxisStore[4].Axis[15].Pos1.Position := 0.0;
   AxisStore[4].Axis[15].Pos1.Speed := 0;
   AxisStore[4].Axis[15].Pos1.Reached := FALSE;
   AxisStore[4].Axis[15].Pos2.Position := 0.0;
   AxisStore[4].Axis[15].Pos2.Speed := 0;
   AxisStore[4].Axis[15].Pos2.Reached := FALSE;
   AxisStore[4].Axis[15].Pos3.Position := 0.0;
   AxisStore[4].Axis[15].Pos3.Speed := 0;
   AxisStore[4].Axis[15].Pos3.Reached := FALSE;
   AxisStore[4].Axis[15].Pos4.Position := 0.0;
   AxisStore[4].Axis[15].Pos4.Speed := 0;
   AxisStore[4].Axis[15].Pos4.Reached := FALSE;
   AxisStore[4].Axis[15].Pos5.Position := 0.0;
   AxisStore[4].Axis[15].Pos5.Speed := 0;
   AxisStore[4].Axis[15].Pos5.Reached := FALSE;
   AxisStore[4].Axis[15].Pos6.Position := 0.0;
   AxisStore[4].Axis[15].Pos6.Speed := 0;
   AxisStore[4].Axis[15].Pos6.Reached := FALSE;
   AxisStore[4].Axis[15].Pos7.Position := 0.0;
   AxisStore[4].Axis[15].Pos7.Speed := 0;
   AxisStore[4].Axis[15].Pos7.Reached := FALSE;
   AxisStore[4].Axis[15].Pos8.Position := 0.0;
   AxisStore[4].Axis[15].Pos8.Speed := 0;
   AxisStore[4].Axis[15].Pos8.Reached := FALSE;
   AxisStore[4].Axis[15].Pos9.Position := 0.0;
   AxisStore[4].Axis[15].Pos9.Speed := 0;
   AxisStore[4].Axis[15].Pos9.Reached := FALSE;
   AxisStore[4].Axis[15].Pos10.Position := 0.0;
   AxisStore[4].Axis[15].Pos10.Speed := 0;
   AxisStore[4].Axis[15].Pos10.Reached := FALSE;
   AxisStore[4].Axis[15].Pos11.Position := 0.0;
   AxisStore[4].Axis[15].Pos11.Speed := 0;
   AxisStore[4].Axis[15].Pos11.Reached := FALSE;
   AxisStore[4].Axis[15].Pos12.Position := 0.0;
   AxisStore[4].Axis[15].Pos12.Speed := 0;
   AxisStore[4].Axis[15].Pos12.Reached := FALSE;
   AxisStore[4].Axis[15].Pos13.Position := 0.0;
   AxisStore[4].Axis[15].Pos13.Speed := 0;
   AxisStore[4].Axis[15].Pos13.Reached := FALSE;
   AxisStore[4].Axis[15].Pos14.Position := 0.0;
   AxisStore[4].Axis[15].Pos14.Speed := 0;
   AxisStore[4].Axis[15].Pos14.Reached := FALSE;
   AxisStore[4].Axis[15].Pos15.Position := 0.0;
   AxisStore[4].Axis[15].Pos15.Speed := 0;
   AxisStore[4].Axis[15].Pos15.Reached := FALSE;
   AxisStore[4].Axis[15].Pos16.Position := 0.0;
   AxisStore[4].Axis[15].Pos16.Speed := 0;
   AxisStore[4].Axis[15].Pos16.Reached := FALSE;
   AxisStore[4].Axis[15].Pos17.Position := 0.0;
   AxisStore[4].Axis[15].Pos17.Speed := 0;
   AxisStore[4].Axis[15].Pos17.Reached := FALSE;
   AxisStore[4].Axis[15].Pos18.Position := 0.0;
   AxisStore[4].Axis[15].Pos18.Speed := 0;
   AxisStore[4].Axis[15].Pos18.Reached := FALSE;
   AxisStore[4].Axis[15].Pos19.Position := 0.0;
   AxisStore[4].Axis[15].Pos19.Speed := 0;
   AxisStore[4].Axis[15].Pos19.Reached := FALSE;
   AxisStore[4].Axis[15].Pos20.Position := 0.0;
   AxisStore[4].Axis[15].Pos20.Speed := 0;
   AxisStore[4].Axis[15].Pos20.Reached := FALSE;
   AxisStore[4].Axis[15].Pos21.Position := 0.0;
   AxisStore[4].Axis[15].Pos21.Speed := 0;
   AxisStore[4].Axis[15].Pos21.Reached := FALSE;
   AxisStore[4].Axis[15].Pos22.Position := 0.0;
   AxisStore[4].Axis[15].Pos22.Speed := 0;
   AxisStore[4].Axis[15].Pos22.Reached := FALSE;
   AxisStore[4].Axis[15].Pos23.Position := 0.0;
   AxisStore[4].Axis[15].Pos23.Speed := 0;
   AxisStore[4].Axis[15].Pos23.Reached := FALSE;
   AxisStore[4].Axis[15].Pos24.Position := 0.0;
   AxisStore[4].Axis[15].Pos24.Speed := 0;
   AxisStore[4].Axis[15].Pos24.Reached := FALSE;
   AxisStore[4].Axis[15].Pos25.Position := 0.0;
   AxisStore[4].Axis[15].Pos25.Speed := 0;
   AxisStore[4].Axis[15].Pos25.Reached := FALSE;
   AxisStore[4].Axis[15].Pos26.Position := 0.0;
   AxisStore[4].Axis[15].Pos26.Speed := 0;
   AxisStore[4].Axis[15].Pos26.Reached := FALSE;
   AxisStore[4].Axis[15].Pos27.Position := 0.0;
   AxisStore[4].Axis[15].Pos27.Speed := 0;
   AxisStore[4].Axis[15].Pos27.Reached := FALSE;
   AxisStore[4].Axis[15].Pos28.Position := 0.0;
   AxisStore[4].Axis[15].Pos28.Speed := 0;
   AxisStore[4].Axis[15].Pos28.Reached := FALSE;
   AxisStore[4].Axis[15].Pos29.Position := 0.0;
   AxisStore[4].Axis[15].Pos29.Speed := 0;
   AxisStore[4].Axis[15].Pos29.Reached := FALSE;
   AxisStore[4].Axis[15].Pos30.Position := 0.0;
   AxisStore[4].Axis[15].Pos30.Speed := 0;
   AxisStore[4].Axis[15].Pos30.Reached := FALSE;
   AxisStore[5].Axis[1].Pos1.Position := 0.0;
   AxisStore[5].Axis[1].Pos1.Speed := 0;
   AxisStore[5].Axis[1].Pos1.Reached := FALSE;
   AxisStore[5].Axis[1].Pos2.Position := 0.0;
   AxisStore[5].Axis[1].Pos2.Speed := 0;
   AxisStore[5].Axis[1].Pos2.Reached := FALSE;
   AxisStore[5].Axis[1].Pos3.Position := 0.0;
   AxisStore[5].Axis[1].Pos3.Speed := 0;
   AxisStore[5].Axis[1].Pos3.Reached := FALSE;
   AxisStore[5].Axis[1].Pos4.Position := 0.0;
   AxisStore[5].Axis[1].Pos4.Speed := 0;
   AxisStore[5].Axis[1].Pos4.Reached := FALSE;
   AxisStore[5].Axis[1].Pos5.Position := 0.0;
   AxisStore[5].Axis[1].Pos5.Speed := 0;
   AxisStore[5].Axis[1].Pos5.Reached := FALSE;
   AxisStore[5].Axis[1].Pos6.Position := 0.0;
   AxisStore[5].Axis[1].Pos6.Speed := 0;
   AxisStore[5].Axis[1].Pos6.Reached := FALSE;
   AxisStore[5].Axis[1].Pos7.Position := 0.0;
   AxisStore[5].Axis[1].Pos7.Speed := 0;
   AxisStore[5].Axis[1].Pos7.Reached := FALSE;
   AxisStore[5].Axis[1].Pos8.Position := 0.0;
   AxisStore[5].Axis[1].Pos8.Speed := 0;
   AxisStore[5].Axis[1].Pos8.Reached := FALSE;
   AxisStore[5].Axis[1].Pos9.Position := 0.0;
   AxisStore[5].Axis[1].Pos9.Speed := 0;
   AxisStore[5].Axis[1].Pos9.Reached := FALSE;
   AxisStore[5].Axis[1].Pos10.Position := 0.0;
   AxisStore[5].Axis[1].Pos10.Speed := 0;
   AxisStore[5].Axis[1].Pos10.Reached := FALSE;
   AxisStore[5].Axis[1].Pos11.Position := 0.0;
   AxisStore[5].Axis[1].Pos11.Speed := 0;
   AxisStore[5].Axis[1].Pos11.Reached := FALSE;
   AxisStore[5].Axis[1].Pos12.Position := 0.0;
   AxisStore[5].Axis[1].Pos12.Speed := 0;
   AxisStore[5].Axis[1].Pos12.Reached := FALSE;
   AxisStore[5].Axis[1].Pos13.Position := 0.0;
   AxisStore[5].Axis[1].Pos13.Speed := 0;
   AxisStore[5].Axis[1].Pos13.Reached := FALSE;
   AxisStore[5].Axis[1].Pos14.Position := 0.0;
   AxisStore[5].Axis[1].Pos14.Speed := 0;
   AxisStore[5].Axis[1].Pos14.Reached := FALSE;
   AxisStore[5].Axis[1].Pos15.Position := 0.0;
   AxisStore[5].Axis[1].Pos15.Speed := 0;
   AxisStore[5].Axis[1].Pos15.Reached := FALSE;
   AxisStore[5].Axis[1].Pos16.Position := 0.0;
   AxisStore[5].Axis[1].Pos16.Speed := 0;
   AxisStore[5].Axis[1].Pos16.Reached := FALSE;
   AxisStore[5].Axis[1].Pos17.Position := 0.0;
   AxisStore[5].Axis[1].Pos17.Speed := 0;
   AxisStore[5].Axis[1].Pos17.Reached := FALSE;
   AxisStore[5].Axis[1].Pos18.Position := 0.0;
   AxisStore[5].Axis[1].Pos18.Speed := 0;
   AxisStore[5].Axis[1].Pos18.Reached := FALSE;
   AxisStore[5].Axis[1].Pos19.Position := 0.0;
   AxisStore[5].Axis[1].Pos19.Speed := 0;
   AxisStore[5].Axis[1].Pos19.Reached := FALSE;
   AxisStore[5].Axis[1].Pos20.Position := 0.0;
   AxisStore[5].Axis[1].Pos20.Speed := 0;
   AxisStore[5].Axis[1].Pos20.Reached := FALSE;
   AxisStore[5].Axis[1].Pos21.Position := 0.0;
   AxisStore[5].Axis[1].Pos21.Speed := 0;
   AxisStore[5].Axis[1].Pos21.Reached := FALSE;
   AxisStore[5].Axis[1].Pos22.Position := 0.0;
   AxisStore[5].Axis[1].Pos22.Speed := 0;
   AxisStore[5].Axis[1].Pos22.Reached := FALSE;
   AxisStore[5].Axis[1].Pos23.Position := 0.0;
   AxisStore[5].Axis[1].Pos23.Speed := 0;
   AxisStore[5].Axis[1].Pos23.Reached := FALSE;
   AxisStore[5].Axis[1].Pos24.Position := 0.0;
   AxisStore[5].Axis[1].Pos24.Speed := 0;
   AxisStore[5].Axis[1].Pos24.Reached := FALSE;
   AxisStore[5].Axis[1].Pos25.Position := 0.0;
   AxisStore[5].Axis[1].Pos25.Speed := 0;
   AxisStore[5].Axis[1].Pos25.Reached := FALSE;
   AxisStore[5].Axis[1].Pos26.Position := 0.0;
   AxisStore[5].Axis[1].Pos26.Speed := 0;
   AxisStore[5].Axis[1].Pos26.Reached := FALSE;
   AxisStore[5].Axis[1].Pos27.Position := 0.0;
   AxisStore[5].Axis[1].Pos27.Speed := 0;
   AxisStore[5].Axis[1].Pos27.Reached := FALSE;
   AxisStore[5].Axis[1].Pos28.Position := 0.0;
   AxisStore[5].Axis[1].Pos28.Speed := 0;
   AxisStore[5].Axis[1].Pos28.Reached := FALSE;
   AxisStore[5].Axis[1].Pos29.Position := 0.0;
   AxisStore[5].Axis[1].Pos29.Speed := 0;
   AxisStore[5].Axis[1].Pos29.Reached := FALSE;
   AxisStore[5].Axis[1].Pos30.Position := 0.0;
   AxisStore[5].Axis[1].Pos30.Speed := 0;
   AxisStore[5].Axis[1].Pos30.Reached := FALSE;
   AxisStore[5].Axis[2].Pos1.Position := 0.0;
   AxisStore[5].Axis[2].Pos1.Speed := 0;
   AxisStore[5].Axis[2].Pos1.Reached := FALSE;
   AxisStore[5].Axis[2].Pos2.Position := 0.0;
   AxisStore[5].Axis[2].Pos2.Speed := 0;
   AxisStore[5].Axis[2].Pos2.Reached := FALSE;
   AxisStore[5].Axis[2].Pos3.Position := 0.0;
   AxisStore[5].Axis[2].Pos3.Speed := 0;
   AxisStore[5].Axis[2].Pos3.Reached := FALSE;
   AxisStore[5].Axis[2].Pos4.Position := 0.0;
   AxisStore[5].Axis[2].Pos4.Speed := 0;
   AxisStore[5].Axis[2].Pos4.Reached := FALSE;
   AxisStore[5].Axis[2].Pos5.Position := 0.0;
   AxisStore[5].Axis[2].Pos5.Speed := 0;
   AxisStore[5].Axis[2].Pos5.Reached := FALSE;
   AxisStore[5].Axis[2].Pos6.Position := 0.0;
   AxisStore[5].Axis[2].Pos6.Speed := 0;
   AxisStore[5].Axis[2].Pos6.Reached := FALSE;
   AxisStore[5].Axis[2].Pos7.Position := 0.0;
   AxisStore[5].Axis[2].Pos7.Speed := 0;
   AxisStore[5].Axis[2].Pos7.Reached := FALSE;
   AxisStore[5].Axis[2].Pos8.Position := 0.0;
   AxisStore[5].Axis[2].Pos8.Speed := 0;
   AxisStore[5].Axis[2].Pos8.Reached := FALSE;
   AxisStore[5].Axis[2].Pos9.Position := 0.0;
   AxisStore[5].Axis[2].Pos9.Speed := 0;
   AxisStore[5].Axis[2].Pos9.Reached := FALSE;
   AxisStore[5].Axis[2].Pos10.Position := 0.0;
   AxisStore[5].Axis[2].Pos10.Speed := 0;
   AxisStore[5].Axis[2].Pos10.Reached := FALSE;
   AxisStore[5].Axis[2].Pos11.Position := 0.0;
   AxisStore[5].Axis[2].Pos11.Speed := 0;
   AxisStore[5].Axis[2].Pos11.Reached := FALSE;
   AxisStore[5].Axis[2].Pos12.Position := 0.0;
   AxisStore[5].Axis[2].Pos12.Speed := 0;
   AxisStore[5].Axis[2].Pos12.Reached := FALSE;
   AxisStore[5].Axis[2].Pos13.Position := 0.0;
   AxisStore[5].Axis[2].Pos13.Speed := 0;
   AxisStore[5].Axis[2].Pos13.Reached := FALSE;
   AxisStore[5].Axis[2].Pos14.Position := 0.0;
   AxisStore[5].Axis[2].Pos14.Speed := 0;
   AxisStore[5].Axis[2].Pos14.Reached := FALSE;
   AxisStore[5].Axis[2].Pos15.Position := 0.0;
   AxisStore[5].Axis[2].Pos15.Speed := 0;
   AxisStore[5].Axis[2].Pos15.Reached := FALSE;
   AxisStore[5].Axis[2].Pos16.Position := 0.0;
   AxisStore[5].Axis[2].Pos16.Speed := 0;
   AxisStore[5].Axis[2].Pos16.Reached := FALSE;
   AxisStore[5].Axis[2].Pos17.Position := 0.0;
   AxisStore[5].Axis[2].Pos17.Speed := 0;
   AxisStore[5].Axis[2].Pos17.Reached := FALSE;
   AxisStore[5].Axis[2].Pos18.Position := 0.0;
   AxisStore[5].Axis[2].Pos18.Speed := 0;
   AxisStore[5].Axis[2].Pos18.Reached := FALSE;
   AxisStore[5].Axis[2].Pos19.Position := 0.0;
   AxisStore[5].Axis[2].Pos19.Speed := 0;
   AxisStore[5].Axis[2].Pos19.Reached := FALSE;
   AxisStore[5].Axis[2].Pos20.Position := 0.0;
   AxisStore[5].Axis[2].Pos20.Speed := 0;
   AxisStore[5].Axis[2].Pos20.Reached := FALSE;
   AxisStore[5].Axis[2].Pos21.Position := 0.0;
   AxisStore[5].Axis[2].Pos21.Speed := 0;
   AxisStore[5].Axis[2].Pos21.Reached := FALSE;
   AxisStore[5].Axis[2].Pos22.Position := 0.0;
   AxisStore[5].Axis[2].Pos22.Speed := 0;
   AxisStore[5].Axis[2].Pos22.Reached := FALSE;
   AxisStore[5].Axis[2].Pos23.Position := 0.0;
   AxisStore[5].Axis[2].Pos23.Speed := 0;
   AxisStore[5].Axis[2].Pos23.Reached := FALSE;
   AxisStore[5].Axis[2].Pos24.Position := 0.0;
   AxisStore[5].Axis[2].Pos24.Speed := 0;
   AxisStore[5].Axis[2].Pos24.Reached := FALSE;
   AxisStore[5].Axis[2].Pos25.Position := 0.0;
   AxisStore[5].Axis[2].Pos25.Speed := 0;
   AxisStore[5].Axis[2].Pos25.Reached := FALSE;
   AxisStore[5].Axis[2].Pos26.Position := 0.0;
   AxisStore[5].Axis[2].Pos26.Speed := 0;
   AxisStore[5].Axis[2].Pos26.Reached := FALSE;
   AxisStore[5].Axis[2].Pos27.Position := 0.0;
   AxisStore[5].Axis[2].Pos27.Speed := 0;
   AxisStore[5].Axis[2].Pos27.Reached := FALSE;
   AxisStore[5].Axis[2].Pos28.Position := 0.0;
   AxisStore[5].Axis[2].Pos28.Speed := 0;
   AxisStore[5].Axis[2].Pos28.Reached := FALSE;
   AxisStore[5].Axis[2].Pos29.Position := 0.0;
   AxisStore[5].Axis[2].Pos29.Speed := 0;
   AxisStore[5].Axis[2].Pos29.Reached := FALSE;
   AxisStore[5].Axis[2].Pos30.Position := 0.0;
   AxisStore[5].Axis[2].Pos30.Speed := 0;
   AxisStore[5].Axis[2].Pos30.Reached := FALSE;
   AxisStore[5].Axis[3].Pos1.Position := 0.0;
   AxisStore[5].Axis[3].Pos1.Speed := 0;
   AxisStore[5].Axis[3].Pos1.Reached := FALSE;
   AxisStore[5].Axis[3].Pos2.Position := 0.0;
   AxisStore[5].Axis[3].Pos2.Speed := 0;
   AxisStore[5].Axis[3].Pos2.Reached := FALSE;
   AxisStore[5].Axis[3].Pos3.Position := 0.0;
   AxisStore[5].Axis[3].Pos3.Speed := 0;
   AxisStore[5].Axis[3].Pos3.Reached := FALSE;
   AxisStore[5].Axis[3].Pos4.Position := 0.0;
   AxisStore[5].Axis[3].Pos4.Speed := 0;
   AxisStore[5].Axis[3].Pos4.Reached := FALSE;
   AxisStore[5].Axis[3].Pos5.Position := 0.0;
   AxisStore[5].Axis[3].Pos5.Speed := 0;
   AxisStore[5].Axis[3].Pos5.Reached := FALSE;
   AxisStore[5].Axis[3].Pos6.Position := 0.0;
   AxisStore[5].Axis[3].Pos6.Speed := 0;
   AxisStore[5].Axis[3].Pos6.Reached := FALSE;
   AxisStore[5].Axis[3].Pos7.Position := 0.0;
   AxisStore[5].Axis[3].Pos7.Speed := 0;
   AxisStore[5].Axis[3].Pos7.Reached := FALSE;
   AxisStore[5].Axis[3].Pos8.Position := 0.0;
   AxisStore[5].Axis[3].Pos8.Speed := 0;
   AxisStore[5].Axis[3].Pos8.Reached := FALSE;
   AxisStore[5].Axis[3].Pos9.Position := 0.0;
   AxisStore[5].Axis[3].Pos9.Speed := 0;
   AxisStore[5].Axis[3].Pos9.Reached := FALSE;
   AxisStore[5].Axis[3].Pos10.Position := 0.0;
   AxisStore[5].Axis[3].Pos10.Speed := 0;
   AxisStore[5].Axis[3].Pos10.Reached := FALSE;
   AxisStore[5].Axis[3].Pos11.Position := 0.0;
   AxisStore[5].Axis[3].Pos11.Speed := 0;
   AxisStore[5].Axis[3].Pos11.Reached := FALSE;
   AxisStore[5].Axis[3].Pos12.Position := 0.0;
   AxisStore[5].Axis[3].Pos12.Speed := 0;
   AxisStore[5].Axis[3].Pos12.Reached := FALSE;
   AxisStore[5].Axis[3].Pos13.Position := 0.0;
   AxisStore[5].Axis[3].Pos13.Speed := 0;
   AxisStore[5].Axis[3].Pos13.Reached := FALSE;
   AxisStore[5].Axis[3].Pos14.Position := 0.0;
   AxisStore[5].Axis[3].Pos14.Speed := 0;
   AxisStore[5].Axis[3].Pos14.Reached := FALSE;
   AxisStore[5].Axis[3].Pos15.Position := 0.0;
   AxisStore[5].Axis[3].Pos15.Speed := 0;
   AxisStore[5].Axis[3].Pos15.Reached := FALSE;
   AxisStore[5].Axis[3].Pos16.Position := 0.0;
   AxisStore[5].Axis[3].Pos16.Speed := 0;
   AxisStore[5].Axis[3].Pos16.Reached := FALSE;
   AxisStore[5].Axis[3].Pos17.Position := 0.0;
   AxisStore[5].Axis[3].Pos17.Speed := 0;
   AxisStore[5].Axis[3].Pos17.Reached := FALSE;
   AxisStore[5].Axis[3].Pos18.Position := 0.0;
   AxisStore[5].Axis[3].Pos18.Speed := 0;
   AxisStore[5].Axis[3].Pos18.Reached := FALSE;
   AxisStore[5].Axis[3].Pos19.Position := 0.0;
   AxisStore[5].Axis[3].Pos19.Speed := 0;
   AxisStore[5].Axis[3].Pos19.Reached := FALSE;
   AxisStore[5].Axis[3].Pos20.Position := 0.0;
   AxisStore[5].Axis[3].Pos20.Speed := 0;
   AxisStore[5].Axis[3].Pos20.Reached := FALSE;
   AxisStore[5].Axis[3].Pos21.Position := 0.0;
   AxisStore[5].Axis[3].Pos21.Speed := 0;
   AxisStore[5].Axis[3].Pos21.Reached := FALSE;
   AxisStore[5].Axis[3].Pos22.Position := 0.0;
   AxisStore[5].Axis[3].Pos22.Speed := 0;
   AxisStore[5].Axis[3].Pos22.Reached := FALSE;
   AxisStore[5].Axis[3].Pos23.Position := 0.0;
   AxisStore[5].Axis[3].Pos23.Speed := 0;
   AxisStore[5].Axis[3].Pos23.Reached := FALSE;
   AxisStore[5].Axis[3].Pos24.Position := 0.0;
   AxisStore[5].Axis[3].Pos24.Speed := 0;
   AxisStore[5].Axis[3].Pos24.Reached := FALSE;
   AxisStore[5].Axis[3].Pos25.Position := 0.0;
   AxisStore[5].Axis[3].Pos25.Speed := 0;
   AxisStore[5].Axis[3].Pos25.Reached := FALSE;
   AxisStore[5].Axis[3].Pos26.Position := 0.0;
   AxisStore[5].Axis[3].Pos26.Speed := 0;
   AxisStore[5].Axis[3].Pos26.Reached := FALSE;
   AxisStore[5].Axis[3].Pos27.Position := 0.0;
   AxisStore[5].Axis[3].Pos27.Speed := 0;
   AxisStore[5].Axis[3].Pos27.Reached := FALSE;
   AxisStore[5].Axis[3].Pos28.Position := 0.0;
   AxisStore[5].Axis[3].Pos28.Speed := 0;
   AxisStore[5].Axis[3].Pos28.Reached := FALSE;
   AxisStore[5].Axis[3].Pos29.Position := 0.0;
   AxisStore[5].Axis[3].Pos29.Speed := 0;
   AxisStore[5].Axis[3].Pos29.Reached := FALSE;
   AxisStore[5].Axis[3].Pos30.Position := 0.0;
   AxisStore[5].Axis[3].Pos30.Speed := 0;
   AxisStore[5].Axis[3].Pos30.Reached := FALSE;
   AxisStore[5].Axis[4].Pos1.Position := 0.0;
   AxisStore[5].Axis[4].Pos1.Speed := 0;
   AxisStore[5].Axis[4].Pos1.Reached := FALSE;
   AxisStore[5].Axis[4].Pos2.Position := 0.0;
   AxisStore[5].Axis[4].Pos2.Speed := 0;
   AxisStore[5].Axis[4].Pos2.Reached := FALSE;
   AxisStore[5].Axis[4].Pos3.Position := 0.0;
   AxisStore[5].Axis[4].Pos3.Speed := 0;
   AxisStore[5].Axis[4].Pos3.Reached := FALSE;
   AxisStore[5].Axis[4].Pos4.Position := 0.0;
   AxisStore[5].Axis[4].Pos4.Speed := 0;
   AxisStore[5].Axis[4].Pos4.Reached := FALSE;
   AxisStore[5].Axis[4].Pos5.Position := 0.0;
   AxisStore[5].Axis[4].Pos5.Speed := 0;
   AxisStore[5].Axis[4].Pos5.Reached := FALSE;
   AxisStore[5].Axis[4].Pos6.Position := 0.0;
   AxisStore[5].Axis[4].Pos6.Speed := 0;
   AxisStore[5].Axis[4].Pos6.Reached := FALSE;
   AxisStore[5].Axis[4].Pos7.Position := 0.0;
   AxisStore[5].Axis[4].Pos7.Speed := 0;
   AxisStore[5].Axis[4].Pos7.Reached := FALSE;
   AxisStore[5].Axis[4].Pos8.Position := 0.0;
   AxisStore[5].Axis[4].Pos8.Speed := 0;
   AxisStore[5].Axis[4].Pos8.Reached := FALSE;
   AxisStore[5].Axis[4].Pos9.Position := 0.0;
   AxisStore[5].Axis[4].Pos9.Speed := 0;
   AxisStore[5].Axis[4].Pos9.Reached := FALSE;
   AxisStore[5].Axis[4].Pos10.Position := 0.0;
   AxisStore[5].Axis[4].Pos10.Speed := 0;
   AxisStore[5].Axis[4].Pos10.Reached := FALSE;
   AxisStore[5].Axis[4].Pos11.Position := 0.0;
   AxisStore[5].Axis[4].Pos11.Speed := 0;
   AxisStore[5].Axis[4].Pos11.Reached := FALSE;
   AxisStore[5].Axis[4].Pos12.Position := 0.0;
   AxisStore[5].Axis[4].Pos12.Speed := 0;
   AxisStore[5].Axis[4].Pos12.Reached := FALSE;
   AxisStore[5].Axis[4].Pos13.Position := 0.0;
   AxisStore[5].Axis[4].Pos13.Speed := 0;
   AxisStore[5].Axis[4].Pos13.Reached := FALSE;
   AxisStore[5].Axis[4].Pos14.Position := 0.0;
   AxisStore[5].Axis[4].Pos14.Speed := 0;
   AxisStore[5].Axis[4].Pos14.Reached := FALSE;
   AxisStore[5].Axis[4].Pos15.Position := 0.0;
   AxisStore[5].Axis[4].Pos15.Speed := 0;
   AxisStore[5].Axis[4].Pos15.Reached := FALSE;
   AxisStore[5].Axis[4].Pos16.Position := 0.0;
   AxisStore[5].Axis[4].Pos16.Speed := 0;
   AxisStore[5].Axis[4].Pos16.Reached := FALSE;
   AxisStore[5].Axis[4].Pos17.Position := 0.0;
   AxisStore[5].Axis[4].Pos17.Speed := 0;
   AxisStore[5].Axis[4].Pos17.Reached := FALSE;
   AxisStore[5].Axis[4].Pos18.Position := 0.0;
   AxisStore[5].Axis[4].Pos18.Speed := 0;
   AxisStore[5].Axis[4].Pos18.Reached := FALSE;
   AxisStore[5].Axis[4].Pos19.Position := 0.0;
   AxisStore[5].Axis[4].Pos19.Speed := 0;
   AxisStore[5].Axis[4].Pos19.Reached := FALSE;
   AxisStore[5].Axis[4].Pos20.Position := 0.0;
   AxisStore[5].Axis[4].Pos20.Speed := 0;
   AxisStore[5].Axis[4].Pos20.Reached := FALSE;
   AxisStore[5].Axis[4].Pos21.Position := 0.0;
   AxisStore[5].Axis[4].Pos21.Speed := 0;
   AxisStore[5].Axis[4].Pos21.Reached := FALSE;
   AxisStore[5].Axis[4].Pos22.Position := 0.0;
   AxisStore[5].Axis[4].Pos22.Speed := 0;
   AxisStore[5].Axis[4].Pos22.Reached := FALSE;
   AxisStore[5].Axis[4].Pos23.Position := 0.0;
   AxisStore[5].Axis[4].Pos23.Speed := 0;
   AxisStore[5].Axis[4].Pos23.Reached := FALSE;
   AxisStore[5].Axis[4].Pos24.Position := 0.0;
   AxisStore[5].Axis[4].Pos24.Speed := 0;
   AxisStore[5].Axis[4].Pos24.Reached := FALSE;
   AxisStore[5].Axis[4].Pos25.Position := 0.0;
   AxisStore[5].Axis[4].Pos25.Speed := 0;
   AxisStore[5].Axis[4].Pos25.Reached := FALSE;
   AxisStore[5].Axis[4].Pos26.Position := 0.0;
   AxisStore[5].Axis[4].Pos26.Speed := 0;
   AxisStore[5].Axis[4].Pos26.Reached := FALSE;
   AxisStore[5].Axis[4].Pos27.Position := 0.0;
   AxisStore[5].Axis[4].Pos27.Speed := 0;
   AxisStore[5].Axis[4].Pos27.Reached := FALSE;
   AxisStore[5].Axis[4].Pos28.Position := 0.0;
   AxisStore[5].Axis[4].Pos28.Speed := 0;
   AxisStore[5].Axis[4].Pos28.Reached := FALSE;
   AxisStore[5].Axis[4].Pos29.Position := 0.0;
   AxisStore[5].Axis[4].Pos29.Speed := 0;
   AxisStore[5].Axis[4].Pos29.Reached := FALSE;
   AxisStore[5].Axis[4].Pos30.Position := 0.0;
   AxisStore[5].Axis[4].Pos30.Speed := 0;
   AxisStore[5].Axis[4].Pos30.Reached := FALSE;
   AxisStore[5].Axis[5].Pos1.Position := 0.0;
   AxisStore[5].Axis[5].Pos1.Speed := 0;
   AxisStore[5].Axis[5].Pos1.Reached := FALSE;
   AxisStore[5].Axis[5].Pos2.Position := 0.0;
   AxisStore[5].Axis[5].Pos2.Speed := 0;
   AxisStore[5].Axis[5].Pos2.Reached := FALSE;
   AxisStore[5].Axis[5].Pos3.Position := 0.0;
   AxisStore[5].Axis[5].Pos3.Speed := 0;
   AxisStore[5].Axis[5].Pos3.Reached := FALSE;
   AxisStore[5].Axis[5].Pos4.Position := 0.0;
   AxisStore[5].Axis[5].Pos4.Speed := 0;
   AxisStore[5].Axis[5].Pos4.Reached := FALSE;
   AxisStore[5].Axis[5].Pos5.Position := 0.0;
   AxisStore[5].Axis[5].Pos5.Speed := 0;
   AxisStore[5].Axis[5].Pos5.Reached := FALSE;
   AxisStore[5].Axis[5].Pos6.Position := 0.0;
   AxisStore[5].Axis[5].Pos6.Speed := 0;
   AxisStore[5].Axis[5].Pos6.Reached := FALSE;
   AxisStore[5].Axis[5].Pos7.Position := 0.0;
   AxisStore[5].Axis[5].Pos7.Speed := 0;
   AxisStore[5].Axis[5].Pos7.Reached := FALSE;
   AxisStore[5].Axis[5].Pos8.Position := 0.0;
   AxisStore[5].Axis[5].Pos8.Speed := 0;
   AxisStore[5].Axis[5].Pos8.Reached := FALSE;
   AxisStore[5].Axis[5].Pos9.Position := 0.0;
   AxisStore[5].Axis[5].Pos9.Speed := 0;
   AxisStore[5].Axis[5].Pos9.Reached := FALSE;
   AxisStore[5].Axis[5].Pos10.Position := 0.0;
   AxisStore[5].Axis[5].Pos10.Speed := 0;
   AxisStore[5].Axis[5].Pos10.Reached := FALSE;
   AxisStore[5].Axis[5].Pos11.Position := 0.0;
   AxisStore[5].Axis[5].Pos11.Speed := 0;
   AxisStore[5].Axis[5].Pos11.Reached := FALSE;
   AxisStore[5].Axis[5].Pos12.Position := 0.0;
   AxisStore[5].Axis[5].Pos12.Speed := 0;
   AxisStore[5].Axis[5].Pos12.Reached := FALSE;
   AxisStore[5].Axis[5].Pos13.Position := 0.0;
   AxisStore[5].Axis[5].Pos13.Speed := 0;
   AxisStore[5].Axis[5].Pos13.Reached := FALSE;
   AxisStore[5].Axis[5].Pos14.Position := 0.0;
   AxisStore[5].Axis[5].Pos14.Speed := 0;
   AxisStore[5].Axis[5].Pos14.Reached := FALSE;
   AxisStore[5].Axis[5].Pos15.Position := 0.0;
   AxisStore[5].Axis[5].Pos15.Speed := 0;
   AxisStore[5].Axis[5].Pos15.Reached := FALSE;
   AxisStore[5].Axis[5].Pos16.Position := 0.0;
   AxisStore[5].Axis[5].Pos16.Speed := 0;
   AxisStore[5].Axis[5].Pos16.Reached := FALSE;
   AxisStore[5].Axis[5].Pos17.Position := 0.0;
   AxisStore[5].Axis[5].Pos17.Speed := 0;
   AxisStore[5].Axis[5].Pos17.Reached := FALSE;
   AxisStore[5].Axis[5].Pos18.Position := 0.0;
   AxisStore[5].Axis[5].Pos18.Speed := 0;
   AxisStore[5].Axis[5].Pos18.Reached := FALSE;
   AxisStore[5].Axis[5].Pos19.Position := 0.0;
   AxisStore[5].Axis[5].Pos19.Speed := 0;
   AxisStore[5].Axis[5].Pos19.Reached := FALSE;
   AxisStore[5].Axis[5].Pos20.Position := 0.0;
   AxisStore[5].Axis[5].Pos20.Speed := 0;
   AxisStore[5].Axis[5].Pos20.Reached := FALSE;
   AxisStore[5].Axis[5].Pos21.Position := 0.0;
   AxisStore[5].Axis[5].Pos21.Speed := 0;
   AxisStore[5].Axis[5].Pos21.Reached := FALSE;
   AxisStore[5].Axis[5].Pos22.Position := 0.0;
   AxisStore[5].Axis[5].Pos22.Speed := 0;
   AxisStore[5].Axis[5].Pos22.Reached := FALSE;
   AxisStore[5].Axis[5].Pos23.Position := 0.0;
   AxisStore[5].Axis[5].Pos23.Speed := 0;
   AxisStore[5].Axis[5].Pos23.Reached := FALSE;
   AxisStore[5].Axis[5].Pos24.Position := 0.0;
   AxisStore[5].Axis[5].Pos24.Speed := 0;
   AxisStore[5].Axis[5].Pos24.Reached := FALSE;
   AxisStore[5].Axis[5].Pos25.Position := 0.0;
   AxisStore[5].Axis[5].Pos25.Speed := 0;
   AxisStore[5].Axis[5].Pos25.Reached := FALSE;
   AxisStore[5].Axis[5].Pos26.Position := 0.0;
   AxisStore[5].Axis[5].Pos26.Speed := 0;
   AxisStore[5].Axis[5].Pos26.Reached := FALSE;
   AxisStore[5].Axis[5].Pos27.Position := 0.0;
   AxisStore[5].Axis[5].Pos27.Speed := 0;
   AxisStore[5].Axis[5].Pos27.Reached := FALSE;
   AxisStore[5].Axis[5].Pos28.Position := 0.0;
   AxisStore[5].Axis[5].Pos28.Speed := 0;
   AxisStore[5].Axis[5].Pos28.Reached := FALSE;
   AxisStore[5].Axis[5].Pos29.Position := 0.0;
   AxisStore[5].Axis[5].Pos29.Speed := 0;
   AxisStore[5].Axis[5].Pos29.Reached := FALSE;
   AxisStore[5].Axis[5].Pos30.Position := 0.0;
   AxisStore[5].Axis[5].Pos30.Speed := 0;
   AxisStore[5].Axis[5].Pos30.Reached := FALSE;
   AxisStore[5].Axis[6].Pos1.Position := 0.0;
   AxisStore[5].Axis[6].Pos1.Speed := 0;
   AxisStore[5].Axis[6].Pos1.Reached := FALSE;
   AxisStore[5].Axis[6].Pos2.Position := 0.0;
   AxisStore[5].Axis[6].Pos2.Speed := 0;
   AxisStore[5].Axis[6].Pos2.Reached := FALSE;
   AxisStore[5].Axis[6].Pos3.Position := 0.0;
   AxisStore[5].Axis[6].Pos3.Speed := 0;
   AxisStore[5].Axis[6].Pos3.Reached := FALSE;
   AxisStore[5].Axis[6].Pos4.Position := 0.0;
   AxisStore[5].Axis[6].Pos4.Speed := 0;
   AxisStore[5].Axis[6].Pos4.Reached := FALSE;
   AxisStore[5].Axis[6].Pos5.Position := 0.0;
   AxisStore[5].Axis[6].Pos5.Speed := 0;
   AxisStore[5].Axis[6].Pos5.Reached := FALSE;
   AxisStore[5].Axis[6].Pos6.Position := 0.0;
   AxisStore[5].Axis[6].Pos6.Speed := 0;
   AxisStore[5].Axis[6].Pos6.Reached := FALSE;
   AxisStore[5].Axis[6].Pos7.Position := 0.0;
   AxisStore[5].Axis[6].Pos7.Speed := 0;
   AxisStore[5].Axis[6].Pos7.Reached := FALSE;
   AxisStore[5].Axis[6].Pos8.Position := 0.0;
   AxisStore[5].Axis[6].Pos8.Speed := 0;
   AxisStore[5].Axis[6].Pos8.Reached := FALSE;
   AxisStore[5].Axis[6].Pos9.Position := 0.0;
   AxisStore[5].Axis[6].Pos9.Speed := 0;
   AxisStore[5].Axis[6].Pos9.Reached := FALSE;
   AxisStore[5].Axis[6].Pos10.Position := 0.0;
   AxisStore[5].Axis[6].Pos10.Speed := 0;
   AxisStore[5].Axis[6].Pos10.Reached := FALSE;
   AxisStore[5].Axis[6].Pos11.Position := 0.0;
   AxisStore[5].Axis[6].Pos11.Speed := 0;
   AxisStore[5].Axis[6].Pos11.Reached := FALSE;
   AxisStore[5].Axis[6].Pos12.Position := 0.0;
   AxisStore[5].Axis[6].Pos12.Speed := 0;
   AxisStore[5].Axis[6].Pos12.Reached := FALSE;
   AxisStore[5].Axis[6].Pos13.Position := 0.0;
   AxisStore[5].Axis[6].Pos13.Speed := 0;
   AxisStore[5].Axis[6].Pos13.Reached := FALSE;
   AxisStore[5].Axis[6].Pos14.Position := 0.0;
   AxisStore[5].Axis[6].Pos14.Speed := 0;
   AxisStore[5].Axis[6].Pos14.Reached := FALSE;
   AxisStore[5].Axis[6].Pos15.Position := 0.0;
   AxisStore[5].Axis[6].Pos15.Speed := 0;
   AxisStore[5].Axis[6].Pos15.Reached := FALSE;
   AxisStore[5].Axis[6].Pos16.Position := 0.0;
   AxisStore[5].Axis[6].Pos16.Speed := 0;
   AxisStore[5].Axis[6].Pos16.Reached := FALSE;
   AxisStore[5].Axis[6].Pos17.Position := 0.0;
   AxisStore[5].Axis[6].Pos17.Speed := 0;
   AxisStore[5].Axis[6].Pos17.Reached := FALSE;
   AxisStore[5].Axis[6].Pos18.Position := 0.0;
   AxisStore[5].Axis[6].Pos18.Speed := 0;
   AxisStore[5].Axis[6].Pos18.Reached := FALSE;
   AxisStore[5].Axis[6].Pos19.Position := 0.0;
   AxisStore[5].Axis[6].Pos19.Speed := 0;
   AxisStore[5].Axis[6].Pos19.Reached := FALSE;
   AxisStore[5].Axis[6].Pos20.Position := 0.0;
   AxisStore[5].Axis[6].Pos20.Speed := 0;
   AxisStore[5].Axis[6].Pos20.Reached := FALSE;
   AxisStore[5].Axis[6].Pos21.Position := 0.0;
   AxisStore[5].Axis[6].Pos21.Speed := 0;
   AxisStore[5].Axis[6].Pos21.Reached := FALSE;
   AxisStore[5].Axis[6].Pos22.Position := 0.0;
   AxisStore[5].Axis[6].Pos22.Speed := 0;
   AxisStore[5].Axis[6].Pos22.Reached := FALSE;
   AxisStore[5].Axis[6].Pos23.Position := 0.0;
   AxisStore[5].Axis[6].Pos23.Speed := 0;
   AxisStore[5].Axis[6].Pos23.Reached := FALSE;
   AxisStore[5].Axis[6].Pos24.Position := 0.0;
   AxisStore[5].Axis[6].Pos24.Speed := 0;
   AxisStore[5].Axis[6].Pos24.Reached := FALSE;
   AxisStore[5].Axis[6].Pos25.Position := 0.0;
   AxisStore[5].Axis[6].Pos25.Speed := 0;
   AxisStore[5].Axis[6].Pos25.Reached := FALSE;
   AxisStore[5].Axis[6].Pos26.Position := 0.0;
   AxisStore[5].Axis[6].Pos26.Speed := 0;
   AxisStore[5].Axis[6].Pos26.Reached := FALSE;
   AxisStore[5].Axis[6].Pos27.Position := 0.0;
   AxisStore[5].Axis[6].Pos27.Speed := 0;
   AxisStore[5].Axis[6].Pos27.Reached := FALSE;
   AxisStore[5].Axis[6].Pos28.Position := 0.0;
   AxisStore[5].Axis[6].Pos28.Speed := 0;
   AxisStore[5].Axis[6].Pos28.Reached := FALSE;
   AxisStore[5].Axis[6].Pos29.Position := 0.0;
   AxisStore[5].Axis[6].Pos29.Speed := 0;
   AxisStore[5].Axis[6].Pos29.Reached := FALSE;
   AxisStore[5].Axis[6].Pos30.Position := 0.0;
   AxisStore[5].Axis[6].Pos30.Speed := 0;
   AxisStore[5].Axis[6].Pos30.Reached := FALSE;
   AxisStore[5].Axis[7].Pos1.Position := 0.0;
   AxisStore[5].Axis[7].Pos1.Speed := 0;
   AxisStore[5].Axis[7].Pos1.Reached := FALSE;
   AxisStore[5].Axis[7].Pos2.Position := 0.0;
   AxisStore[5].Axis[7].Pos2.Speed := 0;
   AxisStore[5].Axis[7].Pos2.Reached := FALSE;
